					IL_strNCopy(
						SourceStr:= apsElements2[4], 
						DstStr:= ADR(sTemp), 
						CharNum:= 5, 
						strCharFill:= ' ' , 
						MaxLen:= 5);
					{warning 'strNCopy'}					
					//strNCopy(ADR(sTemp), 3, arElements2[4], 3);
		
					//strConcat(ADR(AxesActConfig[k].Firmware), 9, ADR(sTemp));
					IL_CONCAT(ADR(refastAxesActConfig[k].sFirmware), ADR(sTemp), ADR(refastAxesActConfig[k].sFirmware), 9);
					
					//check functional package 
					refastAxesActConfig[k].stFunctionalPackages.bMSP := FALSE;
					refastAxesActConfig[k].stFunctionalPackages.bSRV := FALSE;
					refastAxesActConfig[k].stFunctionalPackages.bSNC := FALSE;
					refastAxesActConfig[k].stFunctionalPackages.bML := FALSE;
					refastAxesActConfig[k].stFunctionalPackages.bMA := FALSE;
					refastAxesActConfig[k].stFunctionalPackages.bTF := FALSE;
					
					IF apsElements2[7]^ = 'MSP' THEN
						refastAxesActConfig[k].stFunctionalPackages.bMSP := TRUE;
					ELSIF apsElements2[7]^ = 'SRV' THEN
						refastAxesActConfig[k].stFunctionalPackages.bSRV := TRUE;
					ELSIF apsElements2[7]^ = 'SNC' THEN
						refastAxesActConfig[k].stFunctionalPackages.bSNC := TRUE;
					END_IF
					
					IF apsElements2[8]^ = 'ML' THEN
						refastAxesActConfig[k].stFunctionalPackages.bML := TRUE;
					ELSIF apsElements2[8]^ = 'MA' THEN
						refastAxesActConfig[k].stFunctionalPackages.bMA := TRUE;
					ELSIF apsElements2[8]^ = 'TF' THEN
						refastAxesActConfig[k].stFunctionalPackages.bTF := TRUE;
					END_IF	
					
					// Check DoubleAxis
					refastAxesActConfig[k].stDoubleAxis.bIsDoubleAxis := FALSE;	
					IF (apsElements2[3]^ = 'MPD') 
						OR (apsElements2[3]^ = 'MPM') THEN		(* 2021-08-03 gt: RDK90 #0124 Placon mit OHNE externe Bremse und neuen Steuerteilen *)
						refastAxesActConfig[k].stDoubleAxis.bIsDoubleAxis := TRUE;
						refastAxesActConfig[k].stDoubleAxis.iLeftAxisAddress := M_GetSercosAdress(apsElements[iMAX_NUM_ELEMENTS_C479*i+4], 1);
						refastAxesActConfig[k].stDoubleAxis.iRightAxisAddress := M_GetSercosAdress(apsElements[iMAX_NUM_ELEMENTS_C479*i+4], 2);
					END_IF
					
					k := k+1;
			
				// no Rexroth IO device and no drive	
				ELSIF NOT (apsElements[iMAX_NUM_ELEMENTS_C479*i+1]^ = '') THEN
					refastSercosIOActConfig[j].bAvailable := TRUE;
					refastSercosIOActConfig[j].iSercosAddress := iSercosAddressTemp;	
	
					//	Präfix noch entfernen !!!
					refastSercosIOActConfig[j].sTypeCode 		:= apsElements[iMAX_NUM_ELEMENTS_C479*i+7]^;
					
					// Where are I/O addresses in C-0-0510
					apiPointerToC510[j] := ADR (aiC510[i+1]);	
					j := j +1;			
				END_IF
			END_IF
		//	i:=i+1;
		//UNTIL( arElements[iMAX_NUM_ELEMENTS_C479*i+1]^ = '' OR i >= MAX_SERCOS_DEVICES )
		//END_REPEAT
		END_FOR

		iState := 50;
		iActNoOfSercosIO := j-1;
		iActNoOfDrives := k-1;
		
		i := 1;
		k := 65;
		j := 0;
		l := 1;


		
(* ################################################################################ *)	
// Sort AxesActConfig by locical address
(* ################################################################################ *)				
	50:
			// real axis configured
			IF aiC484[i] = 8 THEN
				FOR j := 1 TO iMAX_AXES_NUMBER DO
					// if Sercos address is configured copy to temp structure
					IF aiC484[i+1] = refastAxesActConfig[j].iSercosAddress THEN
						astAxesActConfigTmp[(i+1)/2] := refastAxesActConfig[j];
						M_DelStructure(ADR(refastAxesActConfig[j]), SIZEOF(refastAxesActConfig[j]));
						j := iMAX_AXES_NUMBER +1;	// Stop Loop
					END_IF
				END_FOR
			ELSIF  aiC484[i] = 16 THEN
 				astAxesActConfigTmp[(i+1)/2].bVirtualAxis := TRUE;	
			END_IF
						
			IF i < ((2*iMAX_AXES_NUMBER) -1 ) THEN	
				i := i +2;
			ELSE
				FOR j := 1 TO iMAX_AXES_NUMBER DO
					IF refastAxesActConfig[j].bRealAxis THEN
					// Save Sercos Address if drive was found but not configured in C-0-0578	
						refastFoundDrivesError[l].bError := TRUE;
						refastFoundDrivesError[l].iSercosAddress := refastAxesActConfig[j].iSercosAddress;
						refastFoundDrivesError[l].sErrorMessage := 'Axis with sercos adress ';
						sTemp2 := INT_TO_STRING(refastFoundDrivesError[l].iSercosAddress);
						//strConcat(ADR(FoundDrivesError[l].ErrorMessage), SIZEOF(FoundDrivesError[l].ErrorMessage) ,	ADR(strTemp));	
						IL_CONCAT(ADR(refastFoundDrivesError[l].sErrorMessage), ADR(sTemp2), ADR(refastFoundDrivesError[l].sErrorMessage), SIZEOF(refastFoundDrivesError[l].sErrorMessage));				
						sTemp2 := 'found, but not configured with IndraWorks (C-0-0578)';
						//strConcat(ADR	(FoundDrivesError[l].ErrorMessage), SIZEOF(FoundDrivesError[l].ErrorMessage) ,	ADR(strTemp));
						IL_CONCAT(ADR(refastFoundDrivesError[l].sErrorMessage), ADR(sTemp2), ADR(refastFoundDrivesError[l].sErrorMessage), SIZEOF(refastFoundDrivesError[l].sErrorMessage));
						
						IF sDiagMessageInt = '' THEN
							sDiagMessageInt := refastFoundDrivesError[l].sErrorMessage;
						END_IF
						
						ML_SetDiagEntry(
							Severity:= enSeverity, 
							Class:= enClass, 
							Facility:= E_LOG_FACILITY.USER, 
							Code:= wDIAG_CODE, 
							Text:= ADR(refastFoundDrivesError[l].sErrorMessage));
												
						l := l +1;
						bErrorTemp := TRUE;
											
					END_IF
				 	refastAxesActConfig [j] := astAxesActConfigTmp[j];	// copy tmp structure back to origuinal structure
				END_FOR
				iState := 53;
				i := 1;
			END_IF	
		
			IF bErrorTemp THEN
				// If error stop FB
				OUT_ErrorID := 	RESOURCE_ERROR;
				OUT_ErrorIdent.Table :=	USER1_TABLE;       
				OUT_ErrorIdent.Additional1 := 16#F0002;
				OUT_ErrorIdent.Additional2 := 16#F0000;
				
				iState := 998;
			END_IF				

(* ################################################################################ *)	
	// Activate all found axes 
	// necessary to acces S-/P-Parameter
(* ################################################################################ *)	
	53: 
		IF IN_bConfigAxes OR bUpdateFirmware THEN
			REPEAT 	// only new cycle if A24 need to be written
				// activate drive if found on ring
				IF refastAxesActConfig[i].bAvailable THEN 
					stDummyAxis.AxisNo := i;
					iA24 := 0;
					
					IF NOT (iA24 = DWORD_TO_DINT(AxisData[stDummyAxis.AxisNo].dwAxisCondition_i)) THEN		// write A24 only if necessary)
						bExecuteWriteA24 := TRUE;
					END_IF	
				ELSIF aiC484[(2*i)-1] = 8 THEN
					stDummyAxis.AxisNo := i;
					iA24 := 2 ;
					
					IF NOT (iA24 = DWORD_TO_DINT(AxisData[stDummyAxis.AxisNo].dwAxisCondition_i)) THEN		// write A24 only if necessary)
						bExecuteWriteA24 := TRUE;
					END_IF	
				END_IF
						
				fbWriteA24(
					Execute:= bExecuteWriteA24, 
					ParameterNumber:= FP_A_0_0024, 
					Value:= iA24, 
					Axis:= stDummyAxis);	
							
				// NEXT Step
				IF fbWriteA24.Done OR NOT bExecuteWriteA24 THEN	
					bExecuteWriteA24 := FALSE;
					fbWriteA24(
						Execute:= FALSE, 
						Axis:= stDummyAxis );	
					i := i + 1;
				
				// Error	
				ELSIF fbWriteA24.Error THEN
					OUT_ErrorID 	:= fbWriteA24.ErrorID;
					OUT_ErrorIdent 	:= fbWriteA24.ErrorIdent;
					fbWriteA24(Execute	:= FALSE,
								Axis	:= stDummyAxis);
					
					iState 		:= 998;
				END_IF	
			
			
				IF i > iMAX_AXES_NUMBER THEN 
					i := 1;
					iState := 55;
				END_IF
				
			UNTIL bExecuteWriteA24 OR (iState = 55) OR (iState = 998)
			END_REPEAT		
		ELSE
			i := 1;
			iState := 55;
		END_IF
(* ################################################################################ *)	
	// Read name A-0-0002 
(* ################################################################################ *)	
	55:
		REPEAT 	// only new cycle if A-0-0002 needs to be read
			stDummyAxis.AxisNo := i;
		
			bExecuteReadName := (aiC484[2*(i-1)+1] = 8) OR (aiC484[2*(i-1)+1] = 16); // Real (8) and Virtual (16) Axes
			
			fbReadStringParameter(
				Execute:= bExecuteReadName, 
				ParameterNumber:=FP_A_0_0002, 
				Axis:= stDummyAxis, 
				Done=> , 
				Active=> , 
				Error=> , 
				ErrorID=> , 
				ErrorIdent=> , 
				Value=> refastAxesActConfig[i].sName );	
	
			IF NOT fbReadStringParameter.Execute THEN
				refastAxesActConfig[i].sName := '';
			END_IF
				
			IF 	fbReadStringParameter.Done OR NOT bExecuteReadName THEN
				i := i +1 ;
				bExecuteReadName := FALSE;
				
				fbReadStringParameter(
					Execute:= FALSE , 
					ParameterNumber:=FP_A_0_0002 , 
					Axis:= stDummyAxis);
					
				IF i > MB_MAX_AXIS_NUMBER THEN
					i := 1;
					iState := 56;
				END_IF	
				
			ELSIF fbReadStringParameter.Error THEN
					OUT_ErrorID 	:= fbReadStringParameter.ErrorID;
					OUT_ErrorIdent 	:= fbReadStringParameter.ErrorIdent;
					fbReadStringParameter(Execute	:= FALSE,
										Axis	:= stDummyAxis);
					iState 		:= 998;	
			END_IF
	
			
		UNTIL bExecuteReadName OR (iState = 56) OR (iState = 998)
		END_REPEAT	
		
		
(* ################################################################################ *)	
	// Read SerialNo of Drive
(* ################################################################################ *)	
		
	56:
		stDummyAxis.AxisNo := i;
		refastAxesActConfig[i].udiSerialNo := 0;
		
		bExecuteReadSerialNo := (aiC484[2*(i-1)+1] = 8) AND refastAxesActConfig[i].bAvailable;
		
		fbReadListParameter(
			Execute			:= bExecuteReadSerialNo, 
			ParameterNumber	:= GVL_P_Param_ID.FP_P_0_1518, 
			NoOfBytes		:= SIZEOF(audiP1518), 
			ValueAdr		:= ADR(audiP1518), 
			Axis			:= stDummyAxis);	
	
		IF 	fbReadListParameter.Done OR NOT bExecuteReadSerialNo THEN
			IF fbReadListParameter.Done THEN
				refastAxesActConfig[i].udiSerialNo :=	audiP1518[4];	// ELEMENT 4 of P-0-1518
			END_IF
			
			i := i +1 ;
			
			fbReadListParameter(
				Execute:= FALSE , 
				ParameterNumber:= GVL_P_Param_ID.FP_P_0_1518,
				Axis:= stDummyAxis);
				
			IF i >	MB_MAX_AXIS_NUMBER THEN
				i := 1;
				sTemp2 := '';
				iState 		:= 57;
			END_IF	
			
		ELSIF fbReadListParameter.Error THEN
				OUT_ErrorID 	:= fbReadListParameter.ErrorID;
				OUT_ErrorIdent 	:= fbReadListParameter.ErrorIdent;
				fbReadListParameter(Execute	:= FALSE,
									Axis	:= stDummyAxis);
				iState 		:= 998;	
		END_IF

(* ################################################################################ *)	
	// Read Safety Type
(* ################################################################################ *)	
				
	57:
		stDummyAxis.AxisNo := i;
		refastAxesActConfig[i].sSafetyType :=	'';
		sTemp2 := '';
		
		bExecuteReadSafetyType := (aiC484[2*(i-1)+1] = 8) AND refastAxesActConfig[i].bAvailable;
	
		fbReadStringParameter(
			Execute:= bExecuteReadSafetyType , 
			ParameterNumber:= FP_P_0_1520, 
			Axis:= stDummyAxis);	
			
		IF fbReadStringParameter.Done THEN
			sTemp2 := fbReadStringParameter.Value;
		END_IF
						
		IF 	fbReadStringParameter.Done OR NOT bExecuteReadSafetyType THEN
			
			udiNoOfElements := IL_StrSplit(ADR(sTemp2),'-',0,FALSE,ADR(apsElements2),TO_UDINT(SIZEOF(apsElements2) - TO_INT(NOT TO_BOOL(LEN(sTemp2)))) );
		//	IL_StrSplit(ADR(strTemp),'-',0,FALSE,ADR(arElements2),TO_UDINT(SIZEOF(arElements2) - TO_INT(NOT TO_BOOL(LEN(strTemp)))) );
			{warning 'JS: strSplit'}
			//strSplit(ADR(strTemp),CHAR_MINUS,0,FALSE,ADR(arElements));
			 // S4 or L3 or L4 or etc
			IF udiNoOfElements >= 5 THEN 
				refastAxesActConfig[i].sSafetyType  := M_GetSafetyType(apsTypeCodeElements:=apsElements2 , bSecondDoubleAxis:=FALSE );
			ELSE
				refastAxesActConfig[i].sSafetyType  := '';
			END_IF
			
			i := i +1 ;
			sTemp2 := '';
			fbReadStringParameter(
				Execute:= FALSE , 
				ParameterNumber:=FP_P_0_1520 , 
				Axis:= stDummyAxis);
				
			IF i >	MB_MAX_AXIS_NUMBER THEN
				i := 1;	(* 2018-07-03 Kohl: war 0, aber Array mit Index 0 ist nicht zugelassen, deshalb 1 *)
				iState 		:= 59;
			END_IF	
			
		ELSIF fbReadStringParameter.Error THEN
				OUT_ErrorID 	:= fbReadStringParameter.ErrorID;
				OUT_ErrorIdent 	:= fbReadStringParameter.ErrorIdent;
				fbReadStringParameter(Execute	:= FALSE,
									Axis	:= stDummyAxis);
				iState 		:= 998;	
		END_IF
		

(* ################################################################################ *)	
	// Read Firmware directory
(* ################################################################################ *)			
		
//58:
//	// copy to internal variable
//	sFirmwareDirectoryTemp := stDriveFirmwarePath;
//
//	// try to open directory
//	udiDirHandle := SysDirOpen(
//					szDir:=sFirmwareDirectoryTemp , 
//					szDirEntry:= sTemp1, 
//					diMaxDirEntry:= 99  , 
//					pDirInfo:=ADR(ar_stDirInfo) , 
//					pResult:=ADR(udiResultOpen) );
//
//	// directory could be opened 					
//	IF (udiResultOpen = Errors.ERR_OK) THEN
//		// delet structure
//		FOR i := 1 TO MAX_NO_FIRMWARE_FILES DO
//			ar_sFirmwareFiles[i] := '';
//		END_FOR
//		uiNoOfFimrwareFiles := 0;
//		
//		// read all files
//		uiFileNo := 1;
//		udiResultRead := SysDirRead(hDir:=udiDirHandle , szDirEntry:=ar_sFirmwareFiles[uiFileNo] , diMaxDirEntry:= 99, pDirInfo:= 0);
//		REPEAT 
//			udiResultRead := SysDirRead(hDir:=udiDirHandle , szDirEntry:=ar_sFirmwareFiles[uiFileNo] , diMaxDirEntry:= 99, pDirInfo:= 0);
//			
//			//END , no more files available
//			IF (udiResultRead = Errors.ERR_END_OF_OBJECT) THEN
//				ar_sFirmwareFiles[uiFileNo] := '';
//				uiFileNo := uiFileNo -1;
//			ELSE	
//				ar_stFirmwareFilesType[uiFileNo]:=	MO_DUT_funGetFirmwareType(ar_sFirmwareFiles[uiFileNo]);
//				uiFileNo := uiFileNo +1;
//			END_IF	
//			
//		UNTIL (udiResultRead = Errors.ERR_END_OF_OBJECT)
//		END_REPEAT 
//		uiNoOfFirmwareFiles := uiFileNo;
//		SysDirClose(hDir:=udiDirHandle );
//		
//		// finish
//		i := 1;
//		iState 		:= 59;		
//	ELSE	// directory does not exist
//		
//		// create directory
//		udiResutlCreate := SysDirCreate(szDir:=sFirmwareDirectoryTemp);
//		// finish
//		i := 1;
//		iState 		:= 59;		
//	END_IF

(* ################################################################################ *)	
	// Read IP address from drive 
(* ################################################################################ *)			
	59:	
		REPEAT 	// only new cycle if S-0-1020 needs to be read
			stDummyAxis.AxisNo := i;
		
			bExecuteReadName := (aiC484[2*(i-1)+1] = 8) 			// Real (8) 
								AND refastAxesActConfig[i].bAvailable 
								AND (
									(AxisData[stDummyAxis.AxisNo].dwAxisCondition_i = 0)  
									OR (AxisData[stDummyAxis.AxisNo].dwAxisCondition_i = 1) 
									OR (AxisData[stDummyAxis.AxisNo].dwAxisCondition_i = 4) 
									OR (AxisData[stDummyAxis.AxisNo].dwAxisCondition_i = 5)
									OR (AxisData[stDummyAxis.AxisNo].dwAxisCondition_i = 8) 
									OR (AxisData[stDummyAxis.AxisNo].dwAxisCondition_i = 9)
									OR (AxisData[stDummyAxis.AxisNo].dwAxisCondition_i = 12)
									OR (AxisData[stDummyAxis.AxisNo].dwAxisCondition_i = 13)
									);
    
			fbReadListParameter(
				Execute:= bExecuteReadName , 
				ParameterNumber:= FP_S_0_1020 , 
				NoOfBytes:= SIZEOF(abDriveIP) , 
				ValueAdr:= ADR(abDriveIP), 
				Done=> , 
				Active=> , 
				Error=> , 
				ErrorID=> , 
				ErrorIdent=> , 
				NoOfRecBytes=> , 
				Axis:=stDummyAxis );	
							
			IF 	fbReadListParameter.Done OR NOT bExecuteReadName THEN
				IF 	bExecuteReadName THEN			
					refastAxesActConfig[i].sIP := '';
					sTemp2 := BYTE_TO_STRING(abDriveIP[0]) ;
					//strConcat(ADR(AxesActConfig[i].IP), SIZEOF(AxesActConfig[i].IP) ,ADR(strTemp));
					IL_CONCAT(ADR(refastAxesActConfig[i].sIP), ADR(sTemp2), ADR(refastAxesActConfig[i].sIP), SIZEOF(refastAxesActConfig[i].sIP));
					sTemp2 := '.' ;
					IL_CONCAT(ADR(refastAxesActConfig[i].sIP), ADR(sTemp2), ADR(refastAxesActConfig[i].sIP), SIZEOF(refastAxesActConfig[i].sIP));
					sTemp2 := BYTE_TO_STRING(abDriveIP[1]) ;
					IL_CONCAT(ADR(refastAxesActConfig[i].sIP), ADR(sTemp2), ADR(refastAxesActConfig[i].sIP), SIZEOF(refastAxesActConfig[i].sIP));
					sTemp2 := '.' ;
					IL_CONCAT(ADR(refastAxesActConfig[i].sIP), ADR(sTemp2), ADR(refastAxesActConfig[i].sIP), SIZEOF(refastAxesActConfig[i].sIP));
					sTemp2 := BYTE_TO_STRING(abDriveIP[2]) ;
					IL_CONCAT(ADR(refastAxesActConfig[i].sIP), ADR(sTemp2), ADR(refastAxesActConfig[i].sIP), SIZEOF(refastAxesActConfig[i].sIP));
					sTemp2 := '.' ;
					IL_CONCAT(ADR(refastAxesActConfig[i].sIP), ADR(sTemp2), ADR(refastAxesActConfig[i].sIP), SIZEOF(refastAxesActConfig[i].sIP));
					sTemp2 := BYTE_TO_STRING(abDriveIP[3]) ;
					IL_CONCAT(ADR(refastAxesActConfig[i].sIP), ADR(sTemp2), ADR(refastAxesActConfig[i].sIP), SIZEOF(refastAxesActConfig[i].sIP));
				ELSE	
					refastAxesActConfig[i].sIP := '';
				END_IF 
				i := i +1 ;
				bExecuteReadName := FALSE;
				
				fbReadListParameter(
					Execute:= FALSE , 
					ParameterNumber:=FP_S_0_1020 , 
					Axis:= stDummyAxis);
					
				IF i > MB_MAX_AXIS_NUMBER THEN
					i := 0;
					iState := 60;
				END_IF	
				
			ELSIF fbReadListParameter.Error THEN
					OUT_ErrorID 	:= fbReadListParameter.ErrorID;
					OUT_ErrorIdent 	:= fbReadListParameter.ErrorIdent;
					fbReadListParameter(Execute	:= FALSE,
										Axis	:= stDummyAxis);
					iState 		:= 998;	
			END_IF	
		UNTIL bExecuteReadName OR (iState = 60) OR (iState = 998)
		END_REPEAT		
	
		
		
(* ################################################################################ *)	
	// Read ata0b directory
(* ################################################################################ *)			
		
	60:	
		iEntry := 0;
		diMaxEntry := SIZEOF(astDirEntry[iEntry].sEntry);
		Result := SysDirSetCurrent(sPathNameInt);
		hDir := SysDirOpen('', astDirEntry[iEntry].sEntry, diMaxEntry, ADR(dir), ADR(Result));
		iEntry := iEntry + 1;
		WHILE Result = Errors.ERR_OK AND hDir <> RTS_INVALID_HANDLE AND iEntry < iMAX_DIR_ENTRY DO
			diMaxEntry := SIZEOF(astDirEntry[iEntry].sEntry);
			Result := SysDirRead(hDir, astDirEntry[iEntry].sEntry, diMaxEntry, ADR(dir));
			IF (DINT_TO_UDINT(dir.diDirectory) AND DirInfoFlags.DF_DIRECTORY) <> 0 THEN
				astDirEntry[iEntry].bDirectory := TRUE;
			END_IF
			iEntry := iEntry + 1;	
		END_WHILE
		Result := SysDirClose(hDir);
		iEntry := iEntry -2;
		
		
		// create new file or open existing?
		fb_SysFileOpenAsync.stMode := 'rw';

		// 2018-07-03: JK Zählerstart geändert von 1 -> 0, weil im Array schon an der Stelle 0 Informationen stehen		
		FOR i := 0 TO iEntry DO
			IF NOT astDirEntry[i].bDirectory THEN
				IF astDirEntry[i].sEntry = sFILE_NAME THEN
					fb_SysFileOpenAsync.stMode := 'r';
				END_IF
			END_IF
		END_FOR
				
		iState 		:= 65;		
			
		
(* ################################################################################ *)	
	// Open UserDefs.cfg 
(* ################################################################################ *)	
	65:		
		fb_SysFileOpenAsync(
			bEnable:= TRUE, 
			stFileName:= sFILE_AND_PATH, 
			stMode:= , 
			bDone=> , 
			bBusy=> , 
			bError=> , 
			wErrorId=> , 
			hFile=> hCfg);
	
			
		IF fb_SysFileOpenAsync.bDone THEN
			fb_SysFileOpenAsync(
				bEnable:= FALSE);
			sBuffer := '';	
			iState :=70;
		END_IF
	
		// Error	
		IF fb_SysFileOpenAsync.bError THEN
			fb_SysFileOpenAsync(
				bEnable:= FALSE);
			iState :=998;
		END_IF
		
(* ################################################################################ *)	
	// Read UserDefsCfg 
(* ################################################################################ *)	
	70:	// DevicePlcAdd.cfg lesen
		fb_SysFileReadAsync(
			bEnable:= TRUE, 
			hFile:= hCfg, 
			pBuffer:= ADR(sBuffer), 
			dwSize:= INT_TO_DWORD(iFileSize), 
			bDone=> , 
			bBusy=> , 
			bError=> , 
			wErrorId=> , 
			dwRead=> dwReadBytes );
	
		IF fb_SysFileReadAsync.bDone THEN
			fb_SysFileReadAsync(
				bEnable:= FALSE);
			iState := 80;
		END_IF
	
		// Error	
		IF fb_SysFileReadAsync.bError THEN
			fb_SysFileReadAsync(
				bEnable:= FALSE);
			iState :=998;
		END_IF
	
80: // Datei schließen
	fb_SysFileCloseAsync(
		bEnable:= TRUE, 
		hFile:= hCfg, 
		bDone=> , 
		bBusy=> , 
		bError=> , 
		wErrorId=> );

	IF fb_SysFileCloseAsync.bDone THEN
		fb_SysFileCloseAsync(
			bEnable:= FALSE);
		iState :=90;
	END_IF

	// Error	
	IF fb_SysFileCloseAsync.bError THEN
		fb_SysFileCloseAsync(
			bEnable:= FALSE);
		iState :=998;
	END_IF
	
90: // Datei in Array of String kopieren und Formatzeichen löschen
	// split String																//Workaround Defdb00192639, -1 if string is empty					
	udiNoOfElements := IL_StrSplit(ADR(sBuffer),IL_Ascii_to_Char(13),0,FALSE,ADR(apsSplit),TO_UDINT(SIZEOF(apsSplit) - TO_INT(NOT TO_BOOL(LEN(sBuffer)))) ); 
	{warning 'JS: strSplit'}
	//strSplit(ADR(Buffer),13 ,0,FALSE,ADR(arSplit));
	
	sLineFeed := IL_Ascii_to_Char(10);
	iEOF := UDINT_TO_INT(udiNoOfElements);
	
	FOR i := 1 TO UDINT_TO_INT(udiNoOfElements) DO 
		//arStringActCfg[i] := DEL_CHARS(arSplit[i]^, strLineFeed);
		IL_StrTrimAll(SourceStr:=apsSplit[i] , DstStr:=ADR(asStringActCfg[i]) , Char:=sLineFeed , MaxLen:=SIZEOF(apsSplit[i]^)-1 );
	END_FOR
	
	// letzte Zeile löschen
	IF iEOF > 2 THEN
		asStringActCfg[iEOF-1] := ''; 
		iEOF	:= iEOF-2;
	END_IF	
	
	iState := 91;	
	
	
(* ################################################################################ *)	
	// Read Inline IO Config 
(* ################################################################################ *)	
91:	
	fbINLNModuleConfigList(
		Execute:= TRUE, 
		SizeOfModuleConfig:=  SIZEOF(InlineIOCfg), 
		ModuleConfigAdr:= ADR(InlineIOCfg), 
		Done=> , 
		Active=> , 
		Error=> , 
		ErrorID=> , 
		ErrorIdent=> , 
		NoOfModuleConfig=> udiNoOfModuleConfig  );

	
	IF fbINLNModuleConfigList.Done THEN
		FOR i := 1 TO iMAX_INLINE_IO DO	
			IF InlineIOCfg[i].ModuleIdSCN <> 0 THEN
				refastInlineIOActConfig[i].bAvailable := TRUE;
				{warning disable C0196}
				refastInlineIOActConfig[i].eIOType := InlineIOCfg[i].ModuleIdSCN;
				{warning restore C0196}
			END_IF
		END_FOR
		
		fbINLNModuleConfigList(
				Execute:= FALSE );

		i := 1;
		iState := 92;
	ELSIF fbINLNModuleConfigList.Error THEN
		fbINLNModuleConfigList(
				Execute:= FALSE );
		i := 1;		
		iState := 92;
	END_IF

(* ################################################################################ *)	
	// Read S20BK+ ModuleType
(* ################################################################################ *)	
92:	
		stDummyAxis.AxisNo := Objects.SERCOS_ADDRESS_1 + refastSercosIOActConfig[i].iSercosAddress -1;
	
		//SercosIOActConfig[i].TypeCode := DUT_S20Type.S20_UNDEFINED;
		
		// Only with S20 BK+
		bExecuteReadModuleType:= refastSercosIOActConfig[i].bAvailable AND (refastSercosIOActConfig[i].sTypeCode ='R911173318');	
		        
		fbReadListParameter(
			Execute			:= bExecuteReadModuleType, 
			ParameterNumber	:= IL_SIIIElementsToIdn(IL_S_PARAM, 0, 1500, 0, 3),(*= Idn = S-0-1500.0.3*) 			
			NoOfBytes		:= SIZEOF(aliS1500_0_3), 
			ValueAdr		:= ADR(aliS1500_0_3), 
			Axis			:= stDummyAxis);	
	
		IF 	fbReadListParameter.Done OR NOT bExecuteReadModuleType THEN
			IF fbReadListParameter.Done THEN			
				FOR j := 0 TO iMAX_MODULE_ON_SERCOS_IO DO
					refastSercosIOActConfig[i].astIOModule[j].IOType := aliS1500_0_3[j];
					refastSercosIOActConfig[i].astIOModule[j].bAvailable :=  (aliS1500_0_3[j] <> LINT#0);
				END_FOR			
			END_IF
			
			i := i +1 ;	
			fbReadListParameter(
				Execute:= FALSE , 
				Axis:= stDummyAxis);
				
			IF i > iMAX_SERCOS_IO(*MB_MAX_AXIS_NUMBER*) THEN		(* 2018-07-03 Kohl: nun MAX_SERCOS_IO, war MB_MAX_AXIS_NUMBER *)
				i := 1;
				sTemp2 := '';
				iState 		:= 99;
			END_IF	
			
		ELSIF fbReadListParameter.Error THEN
				OUT_ErrorID 	:= fbReadListParameter.ErrorID;
				OUT_ErrorIdent 	:= fbReadListParameter.ErrorIdent;
				fbReadListParameter(Execute	:= FALSE,
									Axis	:= stDummyAxis);
				iState 		:= 998;	
		END_IF

(* ################################################################################ *)	
	// End 
(* ################################################################################ *)	
	99:		
		iState := 100;
			
END_CASE
END_METHOD

METHOD M_1ConfigAxes : BOOL

CASE iState OF

	100:
			IF IN_bCheckAxesConfig AND (IN_bConfigAxes OR bUpdateFirmware) THEN 
				iState := 110;
			ELSIF IN_bConfigAxes OR bUpdateFirmware THEN
				i := 1;
				iState := 120;	
			ELSE
				iState := 199;	
			END_IF

(* ################################################################################ *)	
	// Check drive configuration
(* ################################################################################ *)		
	110:
		FOR i := 1 TO iMAX_AXES_NUMBER DO
			// Reset Error structure
			refastAxesConfigError[i].bWrongSercosAddress			:= FALSE;	
			refastAxesConfigError[i].bWrongFirmware 				:= FALSE;
			refastAxesConfigError[i].bWrongFunctionalPackages 		:= FALSE;
			refastAxesConfigError[i].bWrongDoubleAxisConfiguration := FALSE;
			refastAxesConfigError[i].bWrongSafetyType				:= FALSE;
			refastAxesConfigError[i].bDriveFoundAndNotConfigured 	:= FALSE;
			refastAxesConfigError[i].bDriveConfiguredAndNotFound 	:= FALSE;
		
			// Check if found axis = configured axis
			IF  refastAxesActConfig[i].bRealAxis 
				AND refastAxesActConfig[i].bAvailable 
				AND refastAxesCmdConfig[i].bActive THEN
				IF refastAxesActConfig[i].bRealAxis = refastAxesCmdConfig[i].bRealAxis THEN
					// Sercos Address
					IF NOT (refastAxesActConfig[i].iSercosAddress = refastAxesCmdConfig[i].iSercosAddress) THEN
						refastAxesConfigError[i].bWrongSercosAddress := TRUE;
					END_IF
					// Firmware
					IF NOT (LEFT(refastAxesActConfig[i].sFirmware,6) = refastAxesCmdConfig[i].sFirmware) THEN
						refastAxesConfigError[i].bWrongFirmware := TRUE;	
					END_IF  	
					// Functional Packages	
					IF NOT (refastAxesActConfig[i].stFunctionalPackages.bMA = refastAxesCmdConfig[i].stFunctionalPackages.bMA) 
						OR NOT (refastAxesActConfig[i].stFunctionalPackages.bML = refastAxesCmdConfig[i].stFunctionalPackages.bML)
						OR NOT (refastAxesActConfig[i].stFunctionalPackages.bMSP = refastAxesCmdConfig[i].stFunctionalPackages.bMSP)
						OR NOT (refastAxesActConfig[i].stFunctionalPackages.bSNC = refastAxesCmdConfig[i].stFunctionalPackages.bSNC)
						OR NOT (refastAxesActConfig[i].stFunctionalPackages.bSRV = refastAxesCmdConfig[i].stFunctionalPackages.bSRV)
						OR NOT (refastAxesActConfig[i].stFunctionalPackages.bTF = refastAxesCmdConfig[i].stFunctionalPackages.bTF) 
						OR NOT (refastAxesActConfig[i].stFunctionalPackages.bCL = refastAxesCmdConfig[i].stFunctionalPackages.bCL)
						THEN
							refastAxesConfigError[i].bWrongFunctionalPackages := TRUE;	
					END_IF
					// SafetyType
					IF NOT (refastAxesActConfig[i].sSafetyType = refastAxesCmdConfig[i].sSafetyType) THEN
						refastAxesConfigError[i].bWrongSafetyType := TRUE;	
					END_IF  	
					// Double Axis Configuration
					IF NOT (refastAxesActConfig[i].stDoubleAxis.bIsDoubleAxis = refastAxesCmdConfig[i].stDoubleAxis.bIsDoubleAxis)
					OR (
					( NOT (refastAxesActConfig[i].stDoubleAxis.iLeftAxisAddress = refastAxesCmdConfig[i].stDoubleAxis.iLeftAxisAddress)
					OR  NOT (refastAxesActConfig[i].stDoubleAxis.iRightAxisAddress = refastAxesCmdConfig[i].stDoubleAxis.iRightAxisAddress)	
					) AND refastAxesActConfig[i].stDoubleAxis.bIsDoubleAxis AND refastAxesCmdConfig[i].stDoubleAxis.bIsDoubleAxis 					
						) THEN
						refastAxesConfigError[i].bWrongDoubleAxisConfiguration := TRUE;			
					END_IF
				END_IF
			// Found but not configured	
			ELSIF refastAxesActConfig[i].bRealAxis 
				AND refastAxesActConfig[i].bAvailable 
				AND NOT refastAxesCmdConfig[i].bActive THEN
				refastAxesConfigError[i].bDriveFoundAndNotConfigured := TRUE;
			// configured but not found
			ELSIF refastAxesCmdConfig[i].bRealAxis
				AND NOT refastAxesActConfig[i].bAvailable
				AND refastAxesCmdConfig[i].bActive 
				THEN
				refastAxesConfigError[i].bDriveConfiguredAndNotFound := TRUE;
			END_IF
			
			IF refastAxesConfigError[i].bWrongSercosAddress	
				OR refastAxesConfigError[i].bWrongFirmware 
				OR refastAxesConfigError[i].bWrongSafetyType 
				OR refastAxesConfigError[i].bWrongFunctionalPackages 
				OR refastAxesConfigError[i].bWrongDoubleAxisConfiguration
				OR refastAxesConfigError[i].bDriveFoundAndNotConfigured 
				OR refastAxesConfigError[i].bDriveConfiguredAndNotFound THEN
				refastAxesConfigError[i].bError := TRUE;
				bErrorTemp := TRUE;
				
				// Create Error Message
				refastAxesConfigError[i].sErrorMessage := 'Axis ';
				sTemp2 := refastAxesActConfig[i].sName;
				//strConcat(ADR	(AxesConfigError[i].ErrorMessage), SIZEOF(AxesConfigError[i].ErrorMessage) ,	ADR(strTemp));
				IL_CONCAT(ADR(refastAxesConfigError[i].sErrorMessage), ADR(sTemp2), ADR(refastAxesConfigError[i].sErrorMessage), SIZEOF(refastAxesConfigError[i].sErrorMessage));
				sTemp2 := ' with sercos address ';
				IL_CONCAT(ADR(refastAxesConfigError[i].sErrorMessage), ADR(sTemp2), ADR(refastAxesConfigError[i].sErrorMessage), SIZEOF(refastAxesConfigError[i].sErrorMessage));
				sTemp2 := INT_TO_STRING(refastAxesActConfig[i].iSercosAddress);
				IL_CONCAT(ADR(refastAxesConfigError[i].sErrorMessage), ADR(sTemp2), ADR(refastAxesConfigError[i].sErrorMessage), SIZEOF(refastAxesConfigError[i].sErrorMessage));
				sTemp2 := ' shows following error(s): ';
				IL_CONCAT(ADR(refastAxesConfigError[i].sErrorMessage), ADR(sTemp2), ADR(refastAxesConfigError[i].sErrorMessage), SIZEOF(refastAxesConfigError[i].sErrorMessage));
				sTemp2 :='';
				
				IF refastAxesConfigError[i].bWrongSercosAddress	THEN
					sTemp2 :='wrong sercos address';
					//strConcat(ADR	(AxesConfigError[i].ErrorMessage), SIZEOF(AxesConfigError[i].ErrorMessage) ,	ADR(strTemp));
					IL_CONCAT(ADR(refastAxesConfigError[i].sErrorMessage), ADR(sTemp2), ADR(refastAxesConfigError[i].sErrorMessage), SIZEOF(refastAxesConfigError[i].sErrorMessage));
					sTemp2 :=', ';
				END_IF
					
				IF refastAxesConfigError[i].bWrongFirmware	THEN
					//strConcat(ADR	(AxesConfigError[i].ErrorMessage), SIZEOF(AxesConfigError[i].ErrorMessage) ,	ADR(strTemp));
					IL_CONCAT(ADR(refastAxesConfigError[i].sErrorMessage), ADR(sTemp2), ADR(refastAxesConfigError[i].sErrorMessage), SIZEOF(refastAxesConfigError[i].sErrorMessage));
					sTemp2 :='wrong firmware';
					//strConcat(ADR	(AxesConfigError[i].ErrorMessage), SIZEOF(AxesConfigError[i].ErrorMessage) ,	ADR(strTemp));
					IL_CONCAT(ADR(refastAxesConfigError[i].sErrorMessage), ADR(sTemp2), ADR(refastAxesConfigError[i].sErrorMessage), SIZEOF(refastAxesConfigError[i].sErrorMessage));
					sTemp2 :=', ';
				END_IF
				
				IF refastAxesConfigError[i].bWrongSafetyType	THEN
					//strConcat(ADR	(AxesConfigError[i].ErrorMessage), SIZEOF(AxesConfigError[i].ErrorMessage) ,	ADR(strTemp));
					IL_CONCAT(ADR(refastAxesConfigError[i].sErrorMessage), ADR(sTemp2), ADR(refastAxesConfigError[i].sErrorMessage), SIZEOF(refastAxesConfigError[i].sErrorMessage));
					sTemp2 :='wrong SafetyType';
					//strConcat(ADR	(AxesConfigError[i].ErrorMessage), SIZEOF(AxesConfigError[i].ErrorMessage) ,	ADR(strTemp));
					IL_CONCAT(ADR(refastAxesConfigError[i].sErrorMessage), ADR(sTemp2), ADR(refastAxesConfigError[i].sErrorMessage), SIZEOF(refastAxesConfigError[i].sErrorMessage));
					sTemp2 :=', ';
				END_IF
				
				IF refastAxesConfigError[i].bWrongFunctionalPackages	THEN
					//strConcat(ADR	(AxesConfigError[i].ErrorMessage), SIZEOF(AxesConfigError[i].ErrorMessage) ,	ADR(strTemp));
					IL_CONCAT(ADR(refastAxesConfigError[i].sErrorMessage), ADR(sTemp2), ADR(refastAxesConfigError[i].sErrorMessage), SIZEOF(refastAxesConfigError[i].sErrorMessage));
					sTemp2 :='wrong functional package';
					//strConcat(ADR	(AxesConfigError[i].ErrorMessage), SIZEOF(AxesConfigError[i].ErrorMessage) ,	ADR(strTemp));
					IL_CONCAT(ADR(refastAxesConfigError[i].sErrorMessage), ADR(sTemp2), ADR(refastAxesConfigError[i].sErrorMessage), SIZEOF(refastAxesConfigError[i].sErrorMessage));
					sTemp2 :=', ';
				END_IF
				
				IF refastAxesConfigError[i].bWrongDoubleAxisConfiguration	THEN
					//strConcat(ADR	(AxesConfigError[i].ErrorMessage), SIZEOF(AxesConfigError[i].ErrorMessage) ,	ADR(strTemp));
					IL_CONCAT(ADR(refastAxesConfigError[i].sErrorMessage), ADR(sTemp2), ADR(refastAxesConfigError[i].sErrorMessage), SIZEOF(refastAxesConfigError[i].sErrorMessage));
					sTemp2 :='wrong double axis config';
					//strConcat(ADR	(AxesConfigError[i].ErrorMessage), SIZEOF(AxesConfigError[i].ErrorMessage) ,	ADR(strTemp));
					IL_CONCAT(ADR(refastAxesConfigError[i].sErrorMessage), ADR(sTemp2), ADR(refastAxesConfigError[i].sErrorMessage), SIZEOF(refastAxesConfigError[i].sErrorMessage));
					sTemp2 :=', ';
				END_IF
				
				IF refastAxesConfigError[i].bDriveConfiguredAndNotFound	THEN
					//strConcat(ADR	(AxesConfigError[i].ErrorMessage), SIZEOF(AxesConfigError[i].ErrorMessage) ,	ADR(strTemp));
					IL_CONCAT(ADR(refastAxesConfigError[i].sErrorMessage), ADR(sTemp2), ADR(refastAxesConfigError[i].sErrorMessage), SIZEOF(refastAxesConfigError[i].sErrorMessage));
					sTemp2 :='configured but not found';
					//strConcat(ADR	(AxesConfigError[i].ErrorMessage), SIZEOF(AxesConfigError[i].ErrorMessage) ,	ADR(strTemp));
					IL_CONCAT(ADR(refastAxesConfigError[i].sErrorMessage), ADR(sTemp2), ADR(refastAxesConfigError[i].sErrorMessage), SIZEOF(refastAxesConfigError[i].sErrorMessage));
					sTemp2 :=', ';
				END_IF
				
				IF refastAxesConfigError[i].bDriveFoundAndNotConfigured	THEN
					//strConcat(ADR	(AxesConfigError[i].ErrorMessage), SIZEOF(AxesConfigError[i].ErrorMessage) ,	ADR(strTemp));
					IL_CONCAT(ADR(refastAxesConfigError[i].sErrorMessage), ADR(sTemp2), ADR(refastAxesConfigError[i].sErrorMessage), SIZEOF(refastAxesConfigError[i].sErrorMessage));
					sTemp2 :='found but not configured in DeviceCmdConfig';
					//strConcat(ADR	(AxesConfigError[i].ErrorMessage), SIZEOF(AxesConfigError[i].ErrorMessage) ,	ADR(strTemp));
					IL_CONCAT(ADR(refastAxesConfigError[i].sErrorMessage), ADR(sTemp2), ADR(refastAxesConfigError[i].sErrorMessage), SIZEOF(refastAxesConfigError[i].sErrorMessage));
					sTemp2 :=', ';
				END_IF
					
				ML_SetDiagEntry(
						Severity:= enSeverity, 
						Class:= enClass, 
						Facility:= E_LOG_FACILITY.USER, 
						Code:= wDIAG_CODE, 
						Text:= ADR(refastAxesConfigError[i].sErrorMessage));
						
				IF sDiagMessageInt = '' THEN
					sDiagMessageInt := refastAxesConfigError[i].sErrorMessage;
				END_IF		
			
			END_IF
		END_FOR
		
		IF bErrorTemp THEN
		// If error stop FB
			OUT_ErrorID := 	RESOURCE_ERROR;
			OUT_ErrorIdent.Table :=	USER1_TABLE;       
			OUT_ErrorIdent.Additional1 := 16#F0001;
			OUT_ErrorIdent.Additional2 := 16#F0000;
			
			iState := 998;
		ELSE
		// If no error activate all found drives
			iState := 120;	
			i := 1;
		END_IF
		
(* ################################################################################ *)	
	// Activate all found axes
(* ################################################################################ *)	
	120: 
		REPEAT 		// only new cycle if A24 need to be written
			// activate drive if found on ring
			IF refastAxesActConfig[i].bAvailable THEN 
				stDummyAxis.AxisNo := i;
				CASE refastAxesCmdConfig[i].iStatus OF  			
					0: iA24 := 0;
					1: iA24 := 1;
					2: iA24 := 1;
					
					4: iA24 := 4;
					5: iA24 := 5;
					6: iA24 := 5; 
					
					8: iA24 := 8;
					9: iA24 := 9;
					10: iA24 := 9;
				
					12: iA24 := 12; 
					13: iA24 := 13;
					14: iA24 := 13;
					ELSE
						iA24 := 0;
				END_CASE
				
				IF NOT (iA24 = DWORD_TO_DINT(AxisData[stDummyAxis.AxisNo].dwAxisCondition_i)) THEN		// write A24 only if necessary)
					bExecuteWriteA24 := TRUE;
				END_IF	
			ELSIF aiC484[(2*i)-1] = 8 THEN
				stDummyAxis.AxisNo := i;
				// If drive was not on ring
				IF ((refastAxesCmdConfig[i].iStatus > 3) 
						AND (refastAxesCmdConfig[i].iStatus < 7)) THEN
						//Write A24 if command value decoupling is configured
						iA24 := 6;
				ELSIF ((refastAxesCmdConfig[i].iStatus > 11) 
						AND (refastAxesCmdConfig[i].iStatus < 15)) THEN 
					//Write A24 if command value decoupling is configured in PM
					iA24 := 14;
				ELSIF ((refastAxesCmdConfig[i].iStatus > 7) 
						AND (refastAxesCmdConfig[i].iStatus < 11)) THEN 
					//Deactivate Drive in PM
					iA24 := 10 ;
				ELSIF ((refastAxesCmdConfig[i].iStatus > 0) 
						AND (refastAxesCmdConfig[i].iStatus < 3)) THEN 
					//Deactivate Drive
					iA24 := 2 ;
				ELSE	
					//Deactivate Drive
					iA24 := 2 ;
				END_IF
				
				IF NOT (iA24 = DWORD_TO_DINT(AxisData[stDummyAxis.AxisNo].dwAxisCondition_i)) THEN		// write A24 only if necessary)
					bExecuteWriteA24 := TRUE;
				END_IF	
			END_IF
			
			fbWriteA24(
				Execute:= bExecuteWriteA24, 
				ParameterNumber:= FP_A_0_0024, 
				Value:= iA24, 
				Axis:= stDummyAxis);	
						
			// NEXT Step
			IF fbWriteA24.Done OR NOT bExecuteWriteA24 THEN	
				bExecuteWriteA24 := FALSE;
				fbWriteA24(
					Execute:= FALSE, 
					Axis:= stDummyAxis );	
				i := i + 1;
			
			// Error	
			ELSIF fbWriteA24.Error THEN
				OUT_ErrorID 	:= fbWriteA24.ErrorID;
				OUT_ErrorIdent 	:= fbWriteA24.ErrorIdent;
				fbWriteA24(Execute	:= FALSE,
							Axis	:= stDummyAxis);
				
				iState 		:= 998;
			END_IF	
		
			IF i > iMAX_AXES_NUMBER THEN 
				iState := 130;
			END_IF
			
		UNTIL bExecuteWriteA24 OR (iState = 130) OR (iState = 998)
		END_REPEAT		
130:
(* ################################################################################ *)	
// create String for UserDefs.cfg
(* ################################################################################ *)				
	iLineCfg := 1;
	//	Header
	asStringCmdCfg[iLineCfg] := ';--------------- Sercos IO --------------- ';
	iLineCfg := iLineCfg + 1;	 	// next line
	asStringCmdCfg[iLineCfg] := '[SercosIO.Master.0]';	
	iLineCfg := iLineCfg +1;	 	// next line	
	FOR i := 1 TO iMAX_AXES_NUMBER DO
		IF  refastAxesCmdConfig[i].iSercosAddress <> 0 
		AND (	// Entry only with CSoS Safety Axes
			(refastAxesCmdConfig[i].sSafetyType = 'S0')
		OR 	(refastAxesCmdConfig[i].sSafetyType = 'S4')
		OR 	(refastAxesCmdConfig[i].sSafetyType = 'S5')
		OR 	(refastAxesCmdConfig[i].sSafetyType = 'S6')
		OR 	(refastAxesCmdConfig[i].sSafetyType = 'S3')
		OR 	(refastAxesCmdConfig[i].sSafetyType = 'SD')
			) THEN 
			IF  refastAxesActConfig[i].bAvailable THEN
				asStringCmdCfg[iLineCfg] := '; ';
			ELSE			
				asStringCmdCfg[iLineCfg] := '';
			END_IF	
			
			sTemp2 := 'SlaveDeactAddr = ';
			//strConcat(ADR	(arStringCmdCfg[iLineCfg]), SIZEOF(arStringCmdCfg[iLineCfg]) ,	ADR(strTemp));
			IL_CONCAT(ADR(asStringCmdCfg[iLineCfg]), ADR(sTemp2), ADR(asStringCmdCfg[iLineCfg]), SIZEOF(asStringCmdCfg[iLineCfg]));
			sTemp2 := INT_TO_STRING (refastAxesCmdConfig[i].iSercosAddress);
			//strConcat(ADR	(arStringCmdCfg[iLineCfg]), SIZEOF(arStringCmdCfg[iLineCfg]) ,	ADR(strTemp));
			IL_CONCAT(ADR(asStringCmdCfg[iLineCfg]), ADR(sTemp2), ADR(asStringCmdCfg[iLineCfg]), SIZEOF(asStringCmdCfg[iLineCfg]));

			IF NOT (asStringCmdCfg[iLineCfg]= asStringActCfg[iLineCfg]) THEN
				OUT_bReboot := TRUE;
			END_IF
		
			iLineCfg := iLineCfg +1; 	// next line
		END_IF	
	END_FOR
	// finished
	iState := 199;
	
(* ################################################################################ *)	
	// End
(* ################################################################################ *)			
199: 
	iState := 200;		
	
END_CASE
END_METHOD

METHOD M_2ConfigSercosIO : BOOL

CASE iState OF 

(* ################################################################################ *)	
	// enable SIII Buscoupler 
(* ################################################################################ *)	
	200: 
		M_DelStructure(ADR(sRingString), SIZEOF(sRingString));
		M_DelStructure(ADR(apsElements), SIZEOF(apsElements));	
		M_DelStructure(ADR(refastSercosIOConfigError), SIZEOF(refastSercosIOConfigError));
//		M_DelStructure(ADR(SercosIOCmdConfigError), SIZEOF(SercosIOCmdConfigError));
//		M_DelStructure(ADR(SercosIOActConfig_tmp), SIZEOF(SercosIOActConfig_tmp));	
		M_DelStructure(ADR(abSercosIOFoundInConfig), SIZEOF(abSercosIOFoundInConfig));	
		
		
		IF IN_bConfigSercosIO 
			AND IN_bCheckSercosIOConfig THEN
			iState := 210;			
		ELSIF IN_bConfigSercosIO THEN
			iState := 230;
		ELSIF IN_bCheckSercosIOConfig THEN
			iState := 210;
		ELSIF IN_bWriteSercosIOAddress THEN 
			iState := 290;	
		ELSE
			iState := 299;
		END_IF

(* ################################################################################ *)	
	// validity check if enough IOs are found and configured 
	// Check also correct sercos Adress if WriteSercosIOAddress is not enabled
(* ################################################################################ *)	
	210:
		k := 1;
		bIOFound := FALSE;
		IF NOT IN_bWriteSercosIOAddress THEN
			FOR i := 1 TO iMAX_SERCOS_IO DO	
					
				// Reset Error Struct
				refastSercosIOConfigError[i].bError := FALSE;
				refastSercosIOConfigError[i].sErrorMessage := '';
				refastSercosIOConfigError[i].bIOFoundAndNotConfigured := FALSE;	
				refastSercosIOConfigError[i].bIOConfiguredAndNotFound := FALSE;
				refastSercosIOConfigError[i].bWrongSercosAddress := FALSE;
				refastSercosIOConfigError[i].iSercosAddress := 0;
				refastSercosIOConfigError[i].bWrongIOModuleType := FALSE;
				
				IF NOT (refastSercosIOCmdConfig[i].iSercosAddress = 0) THEN 	
					// search trough ActConfig
					FOR j := 1 TO iMAX_SERCOS_IO DO
						abSercosIOFoundInConfig[i] := FALSE;
						IF refastSercosIOCmdConfig[i].iSercosAddress = refastSercosIOActConfig[j].iSercosAddress THEN
							bIOFound := TRUE;
							abSercosIOFoundInConfig[i] := TRUE;
							astSercosIOActConfigTmp[i] := refastSercosIOActConfig[j];
							IF NOT refastSercosIOCmdConfig[i].bActive AND astSercosIOActConfigTmp[i].bAvailable THEN
		 						refastSercosIOConfigError[i].bIOFoundAndNotConfigured := TRUE;
								refastSercosIOConfigError[i].iSercosAddress := astSercosIOActConfigTmp[i].iSercosAddress;	
								refastSercosIOConfigError[i].sName := '';	
							//ELSIF SercosIOCmdConfig[i].Active AND NOT SercosIOActConfig_tmp[i].Available THEN
							//	SercosIOConfigError[i].IOConfiguredAndNotFound := TRUE;
							ELSIF refastSercosIOCmdConfig[i].bActive AND astSercosIOActConfigTmp[i].bAvailable THEN
								IF IN_bCheckSercosIOModuleConfig THEN
									// Check if number of found modules = configured modules 
									astSercosIOActConfigTmp[i].uiNoOfIO_Modules := 0;	
									refastSercosIOCmdConfig[i].uiNoOfIOModules := 0;	
									FOR k := 1 TO iMAX_MODULE_ON_SERCOS_IO DO
										// Count configured Modules
										IF refastSercosIOCmdConfig[i].astIOModule[k].bActive THEN	
											refastSercosIOCmdConfig[i].uiNoOfIOModules := refastSercosIOCmdConfig[i].uiNoOfIOModules +1;
										END_IF 
										// Count found Modules
										IF astSercosIOActConfigTmp[i].astIOModule[k].bAvailable THEN	
											astSercosIOActConfigTmp[i].uiNoOfIO_Modules := astSercosIOActConfigTmp[i].uiNoOfIO_Modules +1;
										END_IF
									END_FOR
									IF (refastSercosIOCmdConfig[i].uiNoOfIOModules > astSercosIOActConfigTmp[i].uiNoOfIO_Modules) THEN
										refastSercosIOConfigError[i].bMoreIOModulesConfiguredThanFound := TRUE;
										refastSercosIOConfigError[i].iSercosAddress := refastSercosIOCmdConfig[i].iSercosAddress;
										refastSercosIOConfigError[i].sName := refastSercosIOCmdConfig[i].sName;
									ELSIF (astSercosIOActConfigTmp[i].uiNoOfIO_Modules > refastSercosIOCmdConfig[i].uiNoOfIOModules ) THEN
										refastSercosIOConfigError[i].bMoreIOModulesFoundThanConfigured := TRUE;
										refastSercosIOConfigError[i].iSercosAddress := refastSercosIOCmdConfig[i].iSercosAddress;
										refastSercosIOConfigError[i].sName := refastSercosIOCmdConfig[i].sName;
									ELSE
										refastSercosIOConfigError[i].bMoreIOModulesConfiguredThanFound := FALSE;	
										refastSercosIOConfigError[i].bMoreIOModulesFoundThanConfigured := FALSE;		
									END_IF
									
									// IF number of found modules = configured modules check if type is OK
									IF NOT refastSercosIOConfigError[i].bMoreIOModulesConfiguredThanFound AND NOT refastSercosIOConfigError[i].bMoreIOModulesFoundThanConfigured THEN
										l := 0;
										FOR k := 1 TO iMAX_MODULE_ON_SERCOS_IO DO
											IF astSercosIOActConfigTmp[i].astIOModule[k].bAvailable THEN
												l := l+1;
												WHILE (NOT refastSercosIOCmdConfig[i].astIOModule[l].bActive) AND NOT (l = iMAX_MODULE_ON_SERCOS_IO) DO
													l := l+1;
												END_WHILE
												IF NOT (refastSercosIOCmdConfig[i].astIOModule[l].eIOType = astSercosIOActConfigTmp[i].astIOModule[k].IOType) THEN
													refastSercosIOConfigError[i].astIO_Module[l].bWrongIOType := TRUE;
													refastSercosIOConfigError[i].bWrongIOModuleType := TRUE;
													refastSercosIOConfigError[i].iSercosAddress := refastSercosIOCmdConfig[i].iSercosAddress;
													refastSercosIOConfigError[i].sName := refastSercosIOCmdConfig[i].sName;
												ELSE	
													refastSercosIOConfigError[i].astIO_Module[l].bWrongIOType := FALSE;	
												END_IF
											END_IF
										END_FOR
									END_IF
								END_IF	
							END_IF
							j := iMAX_SERCOS_IO + 1; // Loop END
						END_IF
					END_FOR
					
					// if not found in ActConfig
					IF NOT bIOFound AND refastSercosIOCmdConfig[i].bActive THEN
						refastSercosIOConfigError[i].bIOConfiguredAndNotFound := TRUE;
						refastSercosIOConfigError[i].iSercosAddress := refastSercosIOCmdConfig[i].iSercosAddress;
						refastSercosIOConfigError[i].sName := refastSercosIOCmdConfig[i].sName;	
					END_IF
					bIOFound := FALSE;
				END_IF	
			END_FOR
		END_IF

		// to have same index like SercosIOCmdConfig
		FOR i := 1 TO iMAX_SERCOS_IO DO
			refastSercosIOActConfig[i] := astSercosIOActConfigTmp[i];
		END_FOR
		
		iState := 220;	

(* ################################################################################ *)	
	// generate Error if necessary 
(* ################################################################################ *)	
	220:
		FOR i := 1 TO iMAX_SERCOS_IO DO
			IF refastSercosIOConfigError[i].bWrongSercosAddress	
				OR refastSercosIOConfigError[i].bIOFoundAndNotConfigured 
				OR refastSercosIOConfigError[i].bIOConfiguredAndNotFound 
				OR refastSercosIOConfigError[i].bMoreIOModulesConfiguredThanFound
				OR refastSercosIOConfigError[i].bMoreIOModulesFoundThanConfigured	 
				OR refastSercosIOConfigError[i].bWrongIOModuleType THEN
					refastSercosIOConfigError[i].bError := TRUE;
									
					bErrorTemp := TRUE;
									
					// Create Error Message
					refastSercosIOConfigError[i].sErrorMessage := 'sercos IO ';
					sTemp2 := refastSercosIOConfigError[i].sName ;
					//strConcat(ADR	(SercosIOConfigError[i].ErrorMessage), SIZEOF(SercosIOConfigError[i].ErrorMessage) ,	ADR(strTemp));
					IL_CONCAT(ADR(refastSercosIOConfigError[i].sErrorMessage), ADR(sTemp2), ADR(refastSercosIOConfigError[i].sErrorMessage), SIZEOF(refastSercosIOConfigError[i].sErrorMessage));
					sTemp2 :=  ' with address '; ;
					//strConcat(ADR	(SercosIOConfigError[i].ErrorMessage), SIZEOF(SercosIOConfigError[i].ErrorMessage) ,	ADR(strTemp));
					IL_CONCAT(ADR(refastSercosIOConfigError[i].sErrorMessage), ADR(sTemp2), ADR(refastSercosIOConfigError[i].sErrorMessage), SIZEOF(refastSercosIOConfigError[i].sErrorMessage));
					sTemp2 := INT_TO_STRING(refastSercosIOConfigError[i].iSercosAddress);
					//strConcat(ADR	(SercosIOConfigError[i].ErrorMessage), SIZEOF(SercosIOConfigError[i].ErrorMessage) ,	ADR(strTemp));
					IL_CONCAT(ADR(refastSercosIOConfigError[i].sErrorMessage), ADR(sTemp2), ADR(refastSercosIOConfigError[i].sErrorMessage), SIZEOF(refastSercosIOConfigError[i].sErrorMessage));
					sTemp2 := ' shows error: ';
					//strConcat(ADR	(SercosIOConfigError[i].ErrorMessage), SIZEOF(SercosIOConfigError[i].ErrorMessage) ,	ADR(strTemp));
					IL_CONCAT(ADR(refastSercosIOConfigError[i].sErrorMessage), ADR(sTemp2), ADR(refastSercosIOConfigError[i].sErrorMessage), SIZEOF(refastSercosIOConfigError[i].sErrorMessage));
					sTemp2 :='';
					IF refastSercosIOConfigError[i].bWrongSercosAddress	THEN
						sTemp2 :='wrong sercos address';
						//strConcat(ADR	(SercosIOConfigError[i].ErrorMessage), SIZEOF(SercosIOConfigError[i].ErrorMessage) ,	ADR(strTemp));
						IL_CONCAT(ADR(refastSercosIOConfigError[i].sErrorMessage), ADR(sTemp2), ADR(refastSercosIOConfigError[i].sErrorMessage), SIZEOF(refastSercosIOConfigError[i].sErrorMessage));
						sTemp2 :=', ';
					END_IF
					
					IF refastSercosIOConfigError[i].bIOConfiguredAndNotFound	THEN
						//strConcat(ADR	(SercosIOConfigError[i].ErrorMessage), SIZEOF(SercosIOConfigError[i].ErrorMessage) ,	ADR(strTemp));
						IL_CONCAT(ADR(refastSercosIOConfigError[i].sErrorMessage), ADR(sTemp2), ADR(refastSercosIOConfigError[i].sErrorMessage), SIZEOF(refastSercosIOConfigError[i].sErrorMessage));
						sTemp2 :='configured but not found';
						//strConcat(ADR	(SercosIOConfigError[i].ErrorMessage), SIZEOF(SercosIOConfigError[i].ErrorMessage) ,	ADR(strTemp));
						IL_CONCAT(ADR(refastSercosIOConfigError[i].sErrorMessage), ADR(sTemp2), ADR(refastSercosIOConfigError[i].sErrorMessage), SIZEOF(refastSercosIOConfigError[i].sErrorMessage));
						sTemp2 :=', ';
					END_IF
					
					IF refastSercosIOConfigError[i].bIOFoundAndNotConfigured	THEN
						//strConcat(ADR	(SercosIOConfigError[i].ErrorMessage), SIZEOF(SercosIOConfigError[i].ErrorMessage) ,	ADR(strTemp));
						IL_CONCAT(ADR(refastSercosIOConfigError[i].sErrorMessage), ADR(sTemp2), ADR(refastSercosIOConfigError[i].sErrorMessage), SIZEOF(refastSercosIOConfigError[i].sErrorMessage));
						sTemp2 :='found but not configured in DeviceCmdConfig';
						//strConcat(ADR	(SercosIOConfigError[i].ErrorMessage), SIZEOF(SercosIOConfigError[i].ErrorMessage) ,	ADR(strTemp));
						IL_CONCAT(ADR(refastSercosIOConfigError[i].sErrorMessage), ADR(sTemp2), ADR(refastSercosIOConfigError[i].sErrorMessage), SIZEOF(refastSercosIOConfigError[i].sErrorMessage));
						sTemp2 :=', ';
					END_IF	
									
					IF refastSercosIOConfigError[i].bMoreIOModulesConfiguredThanFound THEN
						//strConcat(ADR	(SercosIOConfigError[i].ErrorMessage), SIZEOF(SercosIOConfigError[i].ErrorMessage) ,	ADR(strTemp));
						IL_CONCAT(ADR(refastSercosIOConfigError[i].sErrorMessage), ADR(sTemp2), ADR(refastSercosIOConfigError[i].sErrorMessage), SIZEOF(refastSercosIOConfigError[i].sErrorMessage));
						sTemp2 :='more IO Modules configured than found';
						//strConcat(ADR	(SercosIOConfigError[i].ErrorMessage), SIZEOF(SercosIOConfigError[i].ErrorMessage) ,	ADR(strTemp));
						IL_CONCAT(ADR(refastSercosIOConfigError[i].sErrorMessage), ADR(sTemp2), ADR(refastSercosIOConfigError[i].sErrorMessage), SIZEOF(refastSercosIOConfigError[i].sErrorMessage));
						sTemp2 :=', ';
					END_IF	
					
					IF refastSercosIOConfigError[i].bMoreIOModulesFoundThanConfigured THEN
						//strConcat(ADR	(SercosIOConfigError[i].ErrorMessage), SIZEOF(SercosIOConfigError[i].ErrorMessage) ,	ADR(strTemp));
						IL_CONCAT(ADR(refastSercosIOConfigError[i].sErrorMessage), ADR(sTemp2), ADR(refastSercosIOConfigError[i].sErrorMessage), SIZEOF(refastSercosIOConfigError[i].sErrorMessage));
						sTemp2 :='less IO Modules configured than found';
						//strConcat(ADR	(SercosIOConfigError[i].ErrorMessage), SIZEOF(SercosIOConfigError[i].ErrorMessage) ,	ADR(strTemp));
						IL_CONCAT(ADR(refastSercosIOConfigError[i].sErrorMessage), ADR(sTemp2), ADR(refastSercosIOConfigError[i].sErrorMessage), SIZEOF(refastSercosIOConfigError[i].sErrorMessage));
						sTemp2 :=', ';
					END_IF	
					
					IF refastSercosIOConfigError[i].bWrongIOModuleType THEN
						//'wrong IO Module Type: Module 1: expected SSDIxxx - found: SSDOxx ';
						FOR j := 1 TO iMAX_MODULE_ON_SERCOS_IO DO
							IF refastSercosIOConfigError[i].astIO_Module[j].bWrongIOType THEN
								//strConcat(ADR	(SercosIOConfigError[i].ErrorMessage), SIZEOF(SercosIOConfigError[i].ErrorMessage) ,	ADR(strTemp));
								IL_CONCAT(ADR(refastSercosIOConfigError[i].sErrorMessage), ADR(sTemp2), ADR(refastSercosIOConfigError[i].sErrorMessage), SIZEOF(refastSercosIOConfigError[i].sErrorMessage));
								sTemp2 :='wrong IO Module Type: Module ';
								//strConcat(ADR	(SercosIOConfigError[i].ErrorMessage), SIZEOF(SercosIOConfigError[i].ErrorMessage) ,	ADR(strTemp));
								IL_CONCAT(ADR(refastSercosIOConfigError[i].sErrorMessage), ADR(sTemp2), ADR(refastSercosIOConfigError[i].sErrorMessage), SIZEOF(refastSercosIOConfigError[i].sErrorMessage));
								sTemp2 := INT_TO_STRING (j);
								//strConcat(ADR	(SercosIOConfigError[i].ErrorMessage), SIZEOF(SercosIOConfigError[i].ErrorMessage) ,	ADR(strTemp));
								IL_CONCAT(ADR(refastSercosIOConfigError[i].sErrorMessage), ADR(sTemp2), ADR(refastSercosIOConfigError[i].sErrorMessage), SIZEOF(refastSercosIOConfigError[i].sErrorMessage));
								sTemp2 :=': expected: ';
								//strConcat(ADR	(SercosIOConfigError[i].ErrorMessage), SIZEOF(SercosIOConfigError[i].ErrorMessage) ,	ADR(strTemp));
								IL_CONCAT(ADR(refastSercosIOConfigError[i].sErrorMessage), ADR(sTemp2), ADR(refastSercosIOConfigError[i].sErrorMessage), SIZEOF(refastSercosIOConfigError[i].sErrorMessage));
								sTemp2 := M_S20TypeToString(refastSercosIOCmdConfig[i].astIOModule[j].eIOType);
								//strConcat(ADR	(SercosIOConfigError[i].ErrorMessage), SIZEOF(SercosIOConfigError[i].ErrorMessage) ,	ADR(strTemp));
								IL_CONCAT(ADR(refastSercosIOConfigError[i].sErrorMessage), ADR(sTemp2), ADR(refastSercosIOConfigError[i].sErrorMessage), SIZEOF(refastSercosIOConfigError[i].sErrorMessage));
								sTemp2 :=' - found: ';
								//strConcat(ADR	(SercosIOConfigError[i].ErrorMessage), SIZEOF(SercosIOConfigError[i].ErrorMessage) ,	ADR(strTemp));
								IL_CONCAT(ADR(refastSercosIOConfigError[i].sErrorMessage), ADR(sTemp2), ADR(refastSercosIOConfigError[i].sErrorMessage), SIZEOF(refastSercosIOConfigError[i].sErrorMessage));
								sTemp2 := M_S20TypeToString(refastSercosIOActConfig[i].astIOModule[j].IOType);
								//strConcat(ADR	(SercosIOConfigError[i].ErrorMessage), SIZEOF(SercosIOConfigError[i].ErrorMessage) ,	ADR(strTemp));
								IL_CONCAT(ADR(refastSercosIOConfigError[i].sErrorMessage), ADR(sTemp2), ADR(refastSercosIOConfigError[i].sErrorMessage), SIZEOF(refastSercosIOConfigError[i].sErrorMessage));
								sTemp2 :=', ';
							END_IF
						END_FOR
					END_IF	
					
					ML_SetDiagEntry(
						Severity:= enSeverity, 
						Class:= enClass, 
						Facility:= E_LOG_FACILITY.USER, 
						Code:= wDIAG_CODE, 
						Text:= ADR(refastSercosIOConfigError[i].sErrorMessage));
					
					IF sDiagMessageInt = '' THEN
						sDiagMessageInt := refastSercosIOConfigError[i].sErrorMessage;
					END_IF			
						
			END_IF
		END_FOR
			
		IF bErrorTemp THEN  
			OUT_ErrorID := 	RESOURCE_ERROR;
			OUT_ErrorIdent.Table :=	USER1_TABLE;       
			OUT_ErrorIdent.Additional1 := 16#F0003;
			OUT_ErrorIdent.Additional2 := 16#F0000;

			iState 		:= 998;
		ELSIF IN_bConfigSercosIO THEN
			iState 		:= 230;
		ELSIF IN_bWriteSercosIOAddress THEN 
			iState 		:= 290;
		ELSE	
			iState 		:= 299;
		END_IF		
		
		
		
(* ################################################################################ *)	
	// validity check if IO config in C-0-0478 matches to SercosIOCmdConfig
(* ################################################################################ *)		
	230:
		j:= 1;
	
		FOR i := 1 TO iMAX_SERCOS_IO DO
			IF refastSercosIOActConfigC578[i].bAvailable AND (refastSercosIOCmdConfig[i].iSercosAddress <> 0) THEN
				; // OK
				bLoopEnd := FALSE;
				REPEAT
					IF j <= iMAX_SERCOS_IO THEN
						IF refastSercosIOActConfig[i].bAvailable AND refastSercosIOCmdConfig[j].bActive THEN
							astSercosIOActConfigTmp[j].sName := refastSercosIOCmdConfig[j].sName;
							astSercosIOActConfigTmp[j].sTypeCode := refastSercosIOActConfig[i].sTypeCode;
							astSercosIOActConfigTmp[j].astIOModule := refastSercosIOActConfig[i].astIOModule;
							astSercosIOActConfigTmp[j].bAvailable := TRUE;
							astSercosIOActConfigTmp[j].iSercosAddress := refastSercosIOCmdConfig[j].iSercosAddress;
							j := j+1;
							bLoopend := TRUE;
						ELSIF refastSercosIOActConfig[i].bAvailable AND NOT refastSercosIOCmdConfig[j].bActive THEN
							astSercosIOActConfigTmp[j].sName := refastSercosIOCmdConfig[j].sName;
							//SercosIOActConfig_tmp[j].TypeCode := SercosIOActConfig[j].TypeCode;
							astSercosIOActConfigTmp[j].sTypeCode := '';
							astSercosIOActConfigTmp[j].bAvailable := FALSE;
							astSercosIOActConfigTmp[j].iSercosAddress := refastSercosIOCmdConfig[j].iSercosAddress;
							j := j+1;
						ELSIF NOT refastSercosIOActConfig[i].bAvailable AND (refastSercosIOCmdConfig[j].iSercosAddress <> 0) THEN 
							astSercosIOActConfigTmp[j].sName := refastSercosIOCmdConfig[j].sName;
							//SercosIOActConfig_tmp[j].TypeCode := SercosIOActConfig[j].TypeCode;
							astSercosIOActConfigTmp[j].sTypeCode := '';
							astSercosIOActConfigTmp[j].bAvailable := FALSE;
							astSercosIOActConfigTmp[j].iSercosAddress := refastSercosIOCmdConfig[j].iSercosAddress;
							j := j+1;
						ELSE	
							j := j+1;
						END_IF
					ELSE	
						bLoopEnd := TRUE;
					END_IF	
				UNTIL bLoopEnd
				END_REPEAT
				
//			ELSIF NOT	SercosIOActConfigC578[i].Available AND (SercosIOCmdConfig[i].SercosAddress <> 0) THEN
//				; // Too many IO configured in DeviceCmdConfig.sercos_IO
//				SercosIOCmdConfigError.Error := TRUE;
//				SercosIOCmdConfigError.TooManyIOConfigured := TRUE; 
//				SercosIOCmdConfigError.SercosAddress := SercosIOCmdConfig[i].SercosAddress;
//				SercosIOCmdConfigError.Name := SercosIOCmdConfig[i].Name;
//				SercosIOCmdConfigError.ErrorMessage := 'Too many IO stations configured in DeviceCmdConfig.sercos_IO';
//				i := MAX_SERCOS_IO +1; // end loop
//			ELSIF SercosIOActConfigC578[i].Available AND (SercosIOCmdConfig[i].SercosAddress = 0) THEN	
//				; // Too less IO configured in DeviceCmdConfig.sercos_IO
//				SercosIOCmdConfigError.Error := TRUE;
//				SercosIOCmdConfigError.TooLessIOConfigured := TRUE; 
//				SercosIOCmdConfigError.SercosAddress := SercosIOActConfigC578[i].SercosAddress;
//				SercosIOCmdConfigError.ErrorMessage := 'Too less IO stations configured in DeviceCmdConfig.sercos_IO';
//				i := MAX_SERCOS_IO +1; // end loop
			END_IF
			
			// Write Message to MLC Log
//			IF SercosIOCmdConfigError.Error THEN
//				bError_temp := TRUE;	
//				ML_SetDiagEntry(
//					Severity:= enSeverity, 
//					Class:= enClass, 
//					Facility:= E_LOG_FACILITY.USER, 
//					Code:= wDiagCode, 
//					Text:= ADR(SercosIOCmdConfigError.ErrorMessage));
//					
//				IF strDiagMessage_int = '' THEN
//					strDiagMessage_int := SercosIOCmdConfigError.ErrorMessage;
//				END_IF			
//	
//			END_IF
		END_FOR
	
		IF bErrorTemp THEN  
			OUT_ErrorID := 	RESOURCE_ERROR;
			OUT_ErrorIdent.Table :=	USER1_TABLE;       
			OUT_ErrorIdent.Additional1 := 16#F0004;
			OUT_ErrorIdent.Additional2 := 16#F0000;
			iState 		:= 998;
		ELSE	
			M_DelStructure(ADR(refastSercosIOActConfig), SIZEOF(refastSercosIOActConfig));	
			FOR i := 1 TO iMAX_SERCOS_IO DO
				refastSercosIOActConfig[i] := astSercosIOActConfigTmp[i];
			END_FOR
	
			iState 		:= 280;
		END_IF		


(* ################################################################################ *)	
	// Read actual configuration C-0-0578
(* ################################################################################ *)

		
(*		
(* ################################################################################ *)	
	// Read actual configuration C-0-0578
(* ################################################################################ *)			
	235:
		fbReadListParameter(
			Execute			:= TRUE, 
			ParameterNumber	:= GVL_C_Param_ID.FP_C_0_0578, 
			NoOfBytes		:= SIZEOF(sRingString), 
			ValueAdr		:= ADR(sRingString), 
			Axis			:= NoAxis);
			
			IF fbReadListParameter.Done THEN
				fbReadListParameter(Execute	:= FALSE,
									Axis	:= NoAxis);
				iState 	:= 240;
				strSplit(ADR(sRingString),CHAR_COMMA,0,FALSE,ADR(apsElements));
				i 		:= -1;
			ELSIF fbReadListParameter.Error THEN
				ErrorID 	:= fbReadListParameter.ErrorID;
				ErrorIdent 	:= fbReadListParameter.ErrorIdent;
				fbReadListParameter(Execute	:= FALSE,
									Axis	:= NoAxis);
				iState 		:= 998;
			END_IF
		
(* ################################################################################ *)	
	// insert Buscoupler to C-0-0578
(* ################################################################################ *)		
	240:
		REPEAT
			i:= i+1;
				{warning 'weitere R911 Nummern müssen agelegt werden'}
		UNTIL (FUN_TypeCodeIsRexrothIO(TypeCode:=LEFT (apsElements.arWords[uiNumOfElementC578*i+3]^,13)) OR (apsElements.arWords[uiNumOfElementC578*i+3]^ = ''))  
		END_REPEAT
				
		IF i > 0 THEN
			FOR j := 1 TO i DO
				// Build STRING for 1 Axis 
				arAxisString[j] := '';
				// Comma 
				strComma := ',';
				
				//combine Elemenst to C-0-0578
				// example A94,L03100,L05R911173318,'-',NPLC1_E4,S0x00000000,O0x00000008,V94
				//Ax
				strConcat(ADR(arAxisString[j]), SIZEOF(arAxisString[j]), apsElements.arWords[uiNumOfElementC578*(j-1)+1]);
				strConcat(ADR(arAxisString[j]), SIZEOF(arAxisString[j]), ADR(strComma));
				// L03x
				strConcat(ADR(arAxisString[j]), SIZEOF(arAxisString[j]), apsElements.arWords[uiNumOfElementC578*(j-1)+2]);
				strConcat(ADR(arAxisString[j]), SIZEOF(arAxisString[j]), ADR(strComma));
				// L05x
				strConcat(ADR(arAxisString[j]), SIZEOF(arAxisString[j]), apsElements.arWords[uiNumOfElementC578*(j-1)+3]);
				strConcat(ADR(arAxisString[j]), SIZEOF(arAxisString[j]), ADR(strComma));
				// -
				strConcat(ADR(arAxisString[j]), SIZEOF(arAxisString[j]), apsElements.arWords[uiNumOfElementC578*(j-1)+4]);
				strConcat(ADR(arAxisString[j]), SIZEOF(arAxisString[j]), ADR(strComma));
				// Nx
				strConcat(ADR(arAxisString[j]), SIZEOF(arAxisString[j]), apsElements.arWords[uiNumOfElementC578*(j-1)+5]);
				strConcat(ADR(arAxisString[j]), SIZEOF(arAxisString[j]), ADR(strComma));
				// S0x
				strConcat(ADR(arAxisString[j]), SIZEOF(arAxisString[j]), apsElements.arWords[uiNumOfElementC578*(j-1)+6]);
				strConcat(ADR(arAxisString[j]), SIZEOF(arAxisString[j]), ADR(strComma));
				// O0x
				strConcat(ADR(arAxisString[j]), SIZEOF(arAxisString[j]), apsElements.arWords[uiNumOfElementC578*(j-1)+7]);
				strConcat(ADR(arAxisString[j]), SIZEOF(arAxisString[j]), ADR(strComma));
				// Vx
				strConcat(ADR(arAxisString[j]), SIZEOF(arAxisString[j]), apsElements.arWords[uiNumOfElementC578*(j-1)+8]);
			
			END_FOR
		END_IF	
		
		k := i+1;
		i := i -1;

		iState := 250;
		
(* ################################################################################ *)	
	// Build Axis/Buscoupler strings 
(* ################################################################################ *)			
	250:
		// how many buscoupler in C578?	
		REPEAT
			i:= i+1;
		UNTIL (apsElements.arWords[uiNumOfElementC578*i+3]^ = '')  
		END_REPEAT
	
				
		FOR j := k TO i DO   
				//Delete 'A' at beginning of String
			IF (apsElements.arWords[uiNumOfElementC578*(j-1)+1]^ <> '') THEN
				ptString := apsElements.arWords[uiNumOfElementC578*(j-1)+1]+1;
			ELSE
				ptString := apsElements.arWords[uiNumOfElementC578*(j-1)+1];
			END_IF
			
			iSercosAddressTemp :=  STRING_TO_INT(ptString^);	
			
			// Check if IO in SercosIOCmdConfig and set Status depending SercosIOCmdConfig.Active
			FOR l := 1 TO MAX_SERCOS_IO DO
				IF SercosIOCmdConfig[l].SercosAddress = iSercosAddressTemp THEN
					// Build String for C578	
					arAxisString[j] := '';
					// Comma 
					strComma := ',';
	
					//combine Elemenst to C-0-0578
					// example A94,L03100,L05R911173318,'-',NPLC1_E4,S0x00000000,O0x00000008,V94
					//Ax
					strConcat(ADR(arAxisString[j]), SIZEOF(arAxisString[j]), apsElements.arWords[uiNumOfElementC578*(j-1)+1]);
					strConcat(ADR(arAxisString[j]), SIZEOF(arAxisString[j]), ADR(strComma));
					// L03x
					strConcat(ADR(arAxisString[j]), SIZEOF(arAxisString[j]), apsElements.arWords[uiNumOfElementC578*(j-1)+2]);
					strConcat(ADR(arAxisString[j]), SIZEOF(arAxisString[j]), ADR(strComma));
					// L05x
					strConcat(ADR(arAxisString[j]), SIZEOF(arAxisString[j]), apsElements.arWords[uiNumOfElementC578*(j-1)+3]);
					strConcat(ADR(arAxisString[j]), SIZEOF(arAxisString[j]), ADR(strComma));
					// -
					strConcat(ADR(arAxisString[j]), SIZEOF(arAxisString[j]), apsElements.arWords[uiNumOfElementC578*(j-1)+4]);
					strConcat(ADR(arAxisString[j]), SIZEOF(arAxisString[j]), ADR(strComma));
					// N
					strConcat(ADR(arAxisString[j]), SIZEOF(arAxisString[j]), apsElements.arWords[uiNumOfElementC578*(j-1)+5]);
					strConcat(ADR(arAxisString[j]), SIZEOF(arAxisString[j]), ADR(strComma));
					// Status
					IF SercosIOCmdConfig[l].Active THEN
						strTemp := 'S0x00000000';
					ELSE
						strTemp := 'S0x00000002';
					END_IF
					strConcat(ADR(arAxisString[j]), SIZEOF(arAxisString[j]), ADR(strTemp));
					strConcat(ADR(arAxisString[j]), SIZEOF(arAxisString[j]), ADR(strComma));
					// 0Ox
					strConcat(ADR(arAxisString[j]), SIZEOF(arAxisString[j]), apsElements.arWords[uiNumOfElementC578*(j-1)+7]);
					strConcat(ADR(arAxisString[j]), SIZEOF(arAxisString[j]), ADR(strComma));
					// Vx
					strConcat(ADR(arAxisString[j]), SIZEOF(arAxisString[j]), apsElements.arWords[uiNumOfElementC578*(j-1)+5]);
				END_IF
				// End LOOP
				IF SercosIOCmdConfig[l].SercosAddress = 0 THEN 
					l := MAX_SERCOS_IO + 1;
				END_IF
			END_FOR
			
		END_FOR
	
		j := j-1;
		iState := 260;

(* ################################################################################ *)	
	// Build C-0-0578 
(* ################################################################################ *)			
	260:	
		//BUILD C-0-0478
		strC578 :='';
		
		IF j > 0 THEN 
			FOR i := 1 TO j DO
				IF i < j THEN
					strConcat(ADR(strC578), (SIZEOF(strC578)), ADR(arAxisString[i]));
					strConcat(ADR(strC578), (SIZEOF(strC578)), ADR(strComma));
				ELSE	
					strConcat(ADR(strC578), (SIZEOF(strC578)), ADR(arAxisString[i]));
				END_IF
			END_FOR
		END_IF

		iState := 270;


(* ################################################################################ *)	
	// Write C-0-0478
(* ################################################################################ *)			
	270: 
		iState := 280;	
	//	WriteC578(
	//		Execute:= TRUE, 
	//		ParameterNumber:= FP_C_0_0578, 
	//		NoOfBytes:= SIZEOF(strC578), 
	//		ValueAdr:= ADR(strC578), 
	//		Axis:= NoAxis, 
	//		Done=> , 
	//		Active=> );
    //
	//	IF WriteC578.Done THEN
	//		WriteC578(Execute	:= FALSE,
	//				Axis	:= NoAxis);
	//		i		:= 0;
	//				
	//
	//	ELSIF WriteC578.Error THEN
	//		ErrorID 	:= WriteC578.ErrorID;
	//		ErrorIdent 	:= WriteC578.ErrorIdent;
	//		WriteC578(Execute	:= FALSE,
	//							Axis	:= NoAxis);
	//		iState 		:= 998;
	//	END_IF
						
*)		
(* ################################################################################ *)	
// create String for UserDefs.cfg
(* ################################################################################ *)						
	280:
		(* Example:
		;---------- Master.0 ----------
		[SercosIO.Master.0]
		SlaveDeactAddr = 20
		SlaveDeactAddr = 32
		SlaveDeactAddr = 35
		SlaveDeactAddr = 56
		SlaveAddr = 40, DeactModule= 2, 4
		SlaveAddr = 55, DeactLastModules= 3

		;------------------------------
		*)
		IF NOT (iLineCfg > 1) THEN
			//	Header
			asStringCmdCfg[iLineCfg] := ';--------------- Sercos IO --------------- ';
			iLineCfg := iLineCfg + 1;	 	// next line
			asStringCmdCfg[iLineCfg] := '[SercosIO.Master.0]';	
			iLineCfg := iLineCfg +1;	 	// next line
		END_IF
		FOR i := 1 TO iMAX_SERCOS_IO DO
			IF refastSercosIOCmdConfig[i].iSercosAddress <> 0 THEN 
				// deactivate only modules
				IF refastSercosIOCmdConfig[i].bActive THEN
					asStringCmdCfg[iLineCfg] := '';
					bWriteThisLine := FALSE;
					sTemp2 := 'SlaveAddr = ';
					//strConcat(ADR	(arStringCmdCfg[iLineCfg]), SIZEOF(arStringCmdCfg[iLineCfg]) ,	ADR(strTemp));
					IL_CONCAT(ADR(asStringCmdCfg[iLineCfg]), ADR(sTemp2), ADR(asStringCmdCfg[iLineCfg]), SIZEOF(asStringCmdCfg[iLineCfg]));
					sTemp2 := INT_TO_STRING (refastSercosIOCmdConfig[i].iSercosAddress);
					//strConcat(ADR	(arStringCmdCfg[iLineCfg]), SIZEOF(arStringCmdCfg[iLineCfg]) ,	ADR(strTemp));
					IL_CONCAT(ADR(asStringCmdCfg[iLineCfg]), ADR(sTemp2), ADR(asStringCmdCfg[iLineCfg]), SIZEOF(asStringCmdCfg[iLineCfg]));
					sTemp2 :=  ', DeactModule = ';
					//strConcat(ADR	(arStringCmdCfg[iLineCfg]), SIZEOF(arStringCmdCfg[iLineCfg]) ,	ADR(strTemp));
					IL_CONCAT(ADR(asStringCmdCfg[iLineCfg]), ADR(sTemp2), ADR(asStringCmdCfg[iLineCfg]), SIZEOF(asStringCmdCfg[iLineCfg]));
					FOR j := 1 TO iMAX_MODULE_ON_SERCOS_IO DO
						IF NOT refastSercosIOCmdConfig[i].astIOModule[j].bActive AND refastSercosIOCmdConfig[i].astIOModule[j].bConfigured  THEN
							IF bWriteThisLine THEN
								sTemp2 :=  ', ';
								//strConcat(ADR	(arStringCmdCfg[iLineCfg]), SIZEOF(arStringCmdCfg[iLineCfg]) ,	ADR(strTemp));
								IL_CONCAT(ADR(asStringCmdCfg[iLineCfg]), ADR(sTemp2), ADR(asStringCmdCfg[iLineCfg]), SIZEOF(asStringCmdCfg[iLineCfg]));
							END_IF	
							sTemp2 := INT_TO_STRING (j);
							//strConcat(ADR	(arStringCmdCfg[iLineCfg]), SIZEOF(arStringCmdCfg[iLineCfg]) ,	ADR(strTemp));
							IL_CONCAT(ADR(asStringCmdCfg[iLineCfg]), ADR(sTemp2), ADR(asStringCmdCfg[iLineCfg]), SIZEOF(asStringCmdCfg[iLineCfg]));
							
							bWriteThisLine := TRUE;
						END_IF
					END_FOR
				
					
					IF NOT bWriteThisLine THEN
						sTemp2 := 	asStringCmdCfg[iLineCfg];
						asStringCmdCfg[iLineCfg] := '; ';
						//strConcat(ADR (arStringCmdCfg[iLineCfg]), SIZEOF(arStringCmdCfg[iLineCfg]) ,ADR(strTemp));
						IL_CONCAT(ADR(asStringCmdCfg[iLineCfg]), ADR(sTemp2), ADR(asStringCmdCfg[iLineCfg]), SIZEOF(asStringCmdCfg[iLineCfg]));
					END_IF
					
					IF NOT (asStringCmdCfg[iLineCfg]= asStringActCfg[iLineCfg]) THEN
						OUT_bReboot := TRUE;
					END_IF
					iLineCfg := iLineCfg +1; 	// next line
						
				ELSE
					// deactivate complete sercos slave			
					asStringCmdCfg[iLineCfg] := '';
								
					sTemp2 := 'SlaveDeactAddr = ';
					//strConcat(ADR	(arStringCmdCfg[iLineCfg]), SIZEOF(arStringCmdCfg[iLineCfg]) ,	ADR(strTemp));
					IL_CONCAT(ADR(asStringCmdCfg[iLineCfg]), ADR(sTemp2), ADR(asStringCmdCfg[iLineCfg]), SIZEOF(asStringCmdCfg[iLineCfg]));
					sTemp2 := INT_TO_STRING (refastSercosIOCmdConfig[i].iSercosAddress);
					//strConcat(ADR	(arStringCmdCfg[iLineCfg]), SIZEOF(arStringCmdCfg[iLineCfg]) ,	ADR(strTemp));
					IL_CONCAT(ADR(asStringCmdCfg[iLineCfg]), ADR(sTemp2), ADR(asStringCmdCfg[iLineCfg]), SIZEOF(asStringCmdCfg[iLineCfg]));
	
					IF NOT (asStringCmdCfg[iLineCfg]= asStringActCfg[iLineCfg]) THEN
						OUT_bReboot := TRUE;
					END_IF
				
					iLineCfg := iLineCfg +1; 	// next line
				END_IF
			ELSIF refastSercosIOCmdConfig[i].iSercosAddress = 0 THEN
				// End LOOP
	 			i := iMAX_SERCOS_IO + 1;
			END_IF	
		END_FOR
		
		asStringCmdCfg[iLineCfg] := ';-----------------------------------------';
		iLineCfg := iLineCfg +1;	 	// next line

		asStringCmdCfg[iLineCfg] := '';	
		iLineCfg := iLineCfg +1;	 	// next line
		
		iEOF := iLineCfg -1 ;			//End Of File
		
		IF IN_bWriteSercosIOAddress THEN 
			iState 		:= 290;
		ELSE
			iState 		:= 299;
		END_IF
			

(* ################################################################################ *)	
	// Check all I/Os which are found in C-0-0510 (only address of SIII Buscoupler)
(* ################################################################################ *)			
	290: 			
		j := 1;
		FOR i := 1 TO iMAX_SERCOS_IO DO
			refastSercosIOConfigError[i].bError := FALSE;
			refastSercosIOConfigError[i].iSercosAddress := 0;
			refastSercosIOConfigError[i].sErrorMessage := '';
			IF refastSercosIOCmdConfig[i].bActive THEN
				IF NOT (apiPointerToC510[j] = 0) THEN
					apiPointerToC510[j]^ := refastSercosIOCmdConfig[i].iSercosAddress;
					j := j+1;
				ELSE 
					refastSercosIOConfigError[i].bError := TRUE;
					refastSercosIOConfigError[i].iSercosAddress := refastSercosIOCmdConfig[i].iSercosAddress;;
				
					sTemp2 :='';
					refastSercosIOConfigError[i].sErrorMessage := 'IO ';
					sTemp2 := refastSercosIOCmdConfig[i].sName;
					//strConcat(ADR	(SercosIOConfigError[i].ErrorMessage), (SIZEOF(SercosIOConfigError[i].ErrorMessage)) ,	ADR(strTemp));
					IL_CONCAT(ADR(refastSercosIOConfigError[i].sErrorMessage), ADR(sTemp2), ADR(refastSercosIOConfigError[i].sErrorMessage), SIZEOF(refastSercosIOConfigError[i].sErrorMessage));
					sTemp2 := ' with sercos address ';
					//strConcat(ADR	(SercosIOConfigError[i].ErrorMessage), (SIZEOF(SercosIOConfigError[i].ErrorMessage)) ,	ADR(strTemp));
					IL_CONCAT(ADR(refastSercosIOConfigError[i].sErrorMessage), ADR(sTemp2), ADR(refastSercosIOConfigError[i].sErrorMessage), SIZEOF(refastSercosIOConfigError[i].sErrorMessage));
					sTemp2 := INT_TO_STRING(refastSercosIOConfigError[i].iSercosAddress);
					//strConcat(ADR	(SercosIOConfigError[i].ErrorMessage), (SIZEOF(SercosIOConfigError[i].ErrorMessage)) ,	ADR(strTemp));
					IL_CONCAT(ADR(refastSercosIOConfigError[i].sErrorMessage), ADR(sTemp2), ADR(refastSercosIOConfigError[i].sErrorMessage), SIZEOF(refastSercosIOConfigError[i].sErrorMessage));
					sTemp2 := ' not found on bus';				
					IL_CONCAT(ADR(refastSercosIOConfigError[i].sErrorMessage), ADR(sTemp2), ADR(refastSercosIOConfigError[i].sErrorMessage), SIZEOF(refastSercosIOConfigError[i].sErrorMessage));
					bErrorTemp := TRUE;
					
					IF sDiagMessageInt = '' THEN
						sDiagMessageInt := refastSercosIOConfigError[i].sErrorMessage;
					END_IF			
					
				END_IF
			END_IF
		END_FOR
		
		IF bErrorTemp THEN  
			OUT_ErrorID := 	RESOURCE_ERROR;
			OUT_ErrorIdent.Table :=	USER1_TABLE;       
			OUT_ErrorIdent.Additional1 := 16#F0003;
			OUT_ErrorIdent.Additional2 := 16#F0000;
			
			iState 		:= 998;
		ELSE
			iState 		:= 295;
		END_IF	
		
(* ################################################################################ *)	
	// Write C-0-0510 (only address of SIII Buscoupler)
(* ################################################################################ *)					
	295:	
		fbWriteListParameter(
			Execute			:= TRUE, 
			ParameterNumber	:= GVL_C_Param_ID.FP_C_0_0510, 
			NoOfBytes		:= uiLengthArC510, 
			ValueAdr		:= ADR(aiC510), 
			Axis			:= NoAxis );
				
		IF fbWriteListParameter.Done THEN
			fbWriteListParameter(Execute	:= FALSE,
								Axis	:= NoAxis);
			iState 	:= 299;
			i		:= 0;
		ELSIF fbWriteListParameter.Error THEN
			OUT_ErrorID 	:= fbWriteListParameter.ErrorID;
			OUT_ErrorIdent 	:= fbWriteListParameter.ErrorIdent;
			fbWriteListParameter(Execute	:= FALSE,
								Axis	:= NoAxis);
			iState 		:= 998;
		END_IF
	
		
(* ################################################################################ *)	
	// End
(* ################################################################################ *)					
	299:
		iState := 300;		

END_CASE
END_METHOD

METHOD M_3ConfigInlineIO : BOOL

CASE iState OF		
					
	300:
		M_DelStructure(ADR(refastInlineIOConfigError), SIZEOF(refastInlineIOConfigError));
		IF IN_bCheckInlineIOConfig THEN
			iState := 310;
		ELSIF IN_bConfigInlineIO THEN
			iState := 350;
		ELSE
			iState := 399;
		END_IF

(* ################################################################################ *)	
	// Check if Configuration is OK
(* ################################################################################ *)			
	310:
		k:= 1;
		FOR i := 1 TO iMAX_INLINE_IO DO
			IF refastInlineIOActConfig[i].bAvailable THEN	
				refastInlineIOConfigError[i].bIOFoundAndNotConfigured := TRUE;
				refastInlineIOConfigError[i].sName := '';
	
				FOR j := k TO iMAX_INLINE_IO DO
					IF refastInlineIOActConfig[i].bAvailable AND refastInlineIOCmdConfig[j].bActive AND refastInlineIOCmdConfig[j].bConfigured THEN 
						// Wrong IO Type
						IF NOT (refastInlineIOActConfig[i].eIOType = refastInlineIOCmdConfig[j].eIOType) THEN
							refastInlineIOConfigError[i].bWrongIOType := TRUE;
							refastInlineIOConfigError[i].sName := refastInlineIOCmdConfig[j].sName;
						END_IF
						k := j+1;									// save index 
						refastInlineIOConfigError[i].bIOFoundAndNotConfigured := FALSE;
						j := iMAX_SERCOS_IO +1; 		// End LOOP
					END_IF	
				END_FOR
			ELSE	
				i := 	iMAX_SERCOS_IO +1;  // End LOOP
			END_IF	
		END_FOR

	// Are there still some IO configured which where not found on the Inline Bus?
		IF k <= iMAX_INLINE_IO THEN
			FOR j := k TO iMAX_INLINE_IO DO
				IF refastInlineIOCmdConfig[j].bActive THEN
 					refastInlineIOConfigError[j].bIOConfiguredAndNotFound := TRUE;
					refastInlineIOConfigError[j].sName := refastInlineIOCmdConfig[j].sName;
				END_IF
			END_FOR
		END_IF	
	
		iState := 320;
		
(* ################################################################################ *)	
	// generate Error if necessary 
(* ################################################################################ *)	
	320:
		FOR i := 1 TO iMAX_INLINE_IO DO
			IF refastInlineIOConfigError[i].bWrongIOType	
				OR refastInlineIOConfigError[i].bIOFoundAndNotConfigured 
				OR refastInlineIOConfigError[i].bIOConfiguredAndNotFound THEN
					refastInlineIOConfigError[i].bError := TRUE;
									
					bErrorTemp := TRUE;
									
					// Create Error Message
					refastInlineIOConfigError[i].sErrorMessage := 'Inline IO ';
					sTemp2 := refastInlineIOConfigError[i].sName ;
					//strConcat(ADR	(InlineIOConfigError[i].ErrorMessage), SIZEOF(SercosIOConfigError[i].ErrorMessage) ,	ADR(strTemp));
					IL_CONCAT(ADR(refastInlineIOConfigError[i].sErrorMessage), ADR(sTemp2), ADR(refastInlineIOConfigError[i].sErrorMessage), SIZEOF(refastSercosIOConfigError[i].sErrorMessage));
					sTemp2 :=  ' Slot '; ;
					//strConcat(ADR	(InlineIOConfigError[i].ErrorMessage), SIZEOF(InlineIOConfigError[i].ErrorMessage) ,	ADR(strTemp));
					IL_CONCAT(ADR(refastInlineIOConfigError[i].sErrorMessage), ADR(sTemp2), ADR(refastInlineIOConfigError[i].sErrorMessage), SIZEOF(refastSercosIOConfigError[i].sErrorMessage));
					sTemp2 := INT_TO_STRING(i);
					//strConcat(ADR	(InlineIOConfigError[i].ErrorMessage), SIZEOF(InlineIOConfigError[i].ErrorMessage) ,	ADR(strTemp));
					IL_CONCAT(ADR(refastInlineIOConfigError[i].sErrorMessage), ADR(sTemp2), ADR(refastInlineIOConfigError[i].sErrorMessage), SIZEOF(refastSercosIOConfigError[i].sErrorMessage));
					sTemp2 := ' shows error: ';
					//strConcat(ADR	(InlineIOConfigError[i].ErrorMessage), SIZEOF(InlineIOConfigError[i].ErrorMessage) ,	ADR(strTemp));
					IL_CONCAT(ADR(refastInlineIOConfigError[i].sErrorMessage), ADR(sTemp2), ADR(refastInlineIOConfigError[i].sErrorMessage), SIZEOF(refastSercosIOConfigError[i].sErrorMessage));
					sTemp2 :='';
					IF refastInlineIOConfigError[i].bWrongIOType	THEN
						sTemp2 :='wrong IO Type';
						//strConcat(ADR	(InlineIOConfigError[i].ErrorMessage), SIZEOF(InlineIOConfigError[i].ErrorMessage) ,	ADR(strTemp));
						IL_CONCAT(ADR(refastInlineIOConfigError[i].sErrorMessage), ADR(sTemp2), ADR(refastInlineIOConfigError[i].sErrorMessage), SIZEOF(refastSercosIOConfigError[i].sErrorMessage));
						sTemp2 :=', ';
					END_IF
					
					IF refastInlineIOConfigError[i].bIOConfiguredAndNotFound	THEN
						//strConcat(ADR	(InlineIOConfigError[i].ErrorMessage), SIZEOF(InlineIOConfigError[i].ErrorMessage) ,	ADR(strTemp));
						IL_CONCAT(ADR(refastInlineIOConfigError[i].sErrorMessage), ADR(sTemp2), ADR(refastInlineIOConfigError[i].sErrorMessage), SIZEOF(refastSercosIOConfigError[i].sErrorMessage));
						sTemp2 :='configured but not found';
						//strConcat(ADR	(InlineIOConfigError[i].ErrorMessage), SIZEOF(InlineIOConfigError[i].ErrorMessage) ,	ADR(strTemp));
						IL_CONCAT(ADR(refastInlineIOConfigError[i].sErrorMessage), ADR(sTemp2), ADR(refastInlineIOConfigError[i].sErrorMessage), SIZEOF(refastSercosIOConfigError[i].sErrorMessage));
						sTemp2 :=', ';
					END_IF
					
					IF refastInlineIOConfigError[i].bIOFoundAndNotConfigured	THEN
						//strConcat(ADR	(InlineIOConfigError[i].ErrorMessage), SIZEOF(InlineIOConfigError[i].ErrorMessage) ,	ADR(strTemp));
						IL_CONCAT(ADR(refastInlineIOConfigError[i].sErrorMessage), ADR(sTemp2), ADR(refastInlineIOConfigError[i].sErrorMessage), SIZEOF(refastSercosIOConfigError[i].sErrorMessage));
						sTemp2 :='found but not configured in DeviceCmdConfig';
						//strConcat(ADR	(InlineIOConfigError[i].ErrorMessage), SIZEOF(InlineIOConfigError[i].ErrorMessage) ,	ADR(strTemp));
						IL_CONCAT(ADR(refastInlineIOConfigError[i].sErrorMessage), ADR(sTemp2), ADR(refastInlineIOConfigError[i].sErrorMessage), SIZEOF(refastSercosIOConfigError[i].sErrorMessage));
						sTemp2 :=', ';
					END_IF	
					
					ML_SetDiagEntry(
						Severity:= enSeverity, 
						Class:= enClass, 
						Facility:= E_LOG_FACILITY.USER, 
						Code:= wDIAG_CODE, 
						Text:= ADR(refastInlineIOConfigError[i].sErrorMessage));
					
					IF sDiagMessageInt = '' THEN
						sDiagMessageInt := refastInlineIOConfigError[i].sErrorMessage;
					END_IF			
						
			END_IF
		END_FOR
			
		IF bErrorTemp THEN  
			OUT_ErrorID := 	RESOURCE_ERROR;
			OUT_ErrorIdent.Table :=	USER1_TABLE;       
			OUT_ErrorIdent.Additional1 := 16#F0005;
			OUT_ErrorIdent.Additional2 := 16#F0000;

			iState 		:= 998;
		ELSIF IN_bConfigInlineIO THEN
			iState 		:= 350;
		ELSE	
			iState 		:= 399;
		END_IF		
	
			
(* ################################################################################ *)	
	// create String for UserDefs.cfg
(* ################################################################################ *)				
	350:
		(* Example:
	;---------- Master.0 ----------
	[InlineIO.Master.0]
	ModuleDeactPosi = 3
	ModuleDeactPosi = 7
	ModuleDeactPosi = 15
	ModuleDeactPosi = 16
	;------------------------------

		*)

		//	Header
		asStringCmdCfg[iLineCfg] := ';--------------- Inline IO --------------- ';
		iLineCfg := iLineCfg + 1;	 	// next line
		asStringCmdCfg[iLineCfg] := '[InlineIO.Master.0]'	;
		iLineCfg := iLineCfg +1;	 	// next line
		
		FOR i := 1 TO iMAX_INLINE_IO DO
			IF refastInlineIOCmdConfig[i].bConfigured THEN 
				IF refastInlineIOCmdConfig[i].bActive THEN
					asStringCmdCfg[iLineCfg] := '; ';
				ELSE			
					asStringCmdCfg[iLineCfg] := '';
				END_IF	
				
				sTemp2 := 'ModuleDeactPosi = ';
				//strConcat(ADR	(arStringCmdCfg[iLineCfg]), SIZEOF(arStringCmdCfg[iLineCfg]) ,	ADR(strTemp));
				IL_CONCAT(ADR	(asStringCmdCfg[iLineCfg]), ADR(sTemp2), ADR	(asStringCmdCfg[iLineCfg]), SIZEOF(asStringCmdCfg[iLineCfg]));
				sTemp2 := INT_TO_STRING (i);
				//strConcat(ADR	(arStringCmdCfg[iLineCfg]), SIZEOF(arStringCmdCfg[iLineCfg]) ,	ADR(strTemp));
				IL_CONCAT(ADR	(asStringCmdCfg[iLineCfg]), ADR(sTemp2), ADR	(asStringCmdCfg[iLineCfg]), SIZEOF(asStringCmdCfg[iLineCfg]));
				
				IF NOT (asStringCmdCfg[iLineCfg] = asStringActCfg[iLineCfg]) THEN
					OUT_bReboot := TRUE;
				END_IF
			
				iLineCfg := iLineCfg +1; 	// next line
				
			ELSIF NOT refastInlineIOCmdConfig[i].bConfigured  THEN
				// End LOOP
	 			i := iMAX_INLINE_IO + 1;	
			END_IF	
			
			
		END_FOR
		
		asStringCmdCfg[iLineCfg] := ';-----------------------------------------'	;
		iLineCfg := iLineCfg +1;	 	// next line

		asStringCmdCfg[iLineCfg] := ''	;
		iLineCfg := iLineCfg +1;	 	// next line
		
		iEOF := iLineCfg -1 ;			//End Of File
		iState := 399;
		
(* ################################################################################ *)	
	// End
(* ################################################################################ *)					
	399:
		iState := 400;		

END_CASE
END_METHOD

METHOD M_4ConfigProfibsIO : BOOL


CASE iState OF		
(* ################################################################################ *)	
	// create String for UserDefs.cfg
(* ################################################################################ *)						
	400:
		IF IN_bConfigProfibusIO THEN
			iState := 410;
		ELSE
			iState := 499;
		END_IF

	410:
		(* Example:
		; *****************************
		; Onboard Master
		; *****************************
		
		[ProfibusDP.Master.0]
		SlaveDeactAddr = 5
		SlaveDeactAddr = 8
		SlaveDeactAddr = 25
		
		
		; *******************************
		; Master auf einem Funktionsmodul
		; *******************************
		
		[ProfibusDP.Master.1]
		SlaveDeactAddr = 64
		SlaveDeactAddr = 30
		SlaveDeactAddr = 112
		SlaveDeactAddr = 3
	*)

		//	Header

		asStringCmdCfg[iLineCfg] := ';--------------- PROFINET IO --------------- ';
		iLineCfg := iLineCfg + 1;	 	// next line
		
		FOR j := 1 TO iMAX_PROFIBUS_MASTER DO
//			IF ProfibusIOCmdConfig[j,0].Active THEN			// Master is active
				asStringCmdCfg[iLineCfg] := '[ProfibusDP.Master.';
				sTemp2 := INT_TO_STRING(j-1);
				//strConcat(ADR	(arStringCmdCfg[iLineCfg]), SIZEOF(arStringCmdCfg[iLineCfg]) ,	ADR(strTemp));
				IL_CONCAT(ADR(asStringCmdCfg[iLineCfg]), ADR(sTemp2), ADR(asStringCmdCfg[iLineCfg]), SIZEOF(asStringCmdCfg[iLineCfg]));
				sTemp2 := ']';
				//strConcat(ADR	(arStringCmdCfg[iLineCfg]), SIZEOF(arStringCmdCfg[iLineCfg]) ,	ADR(strTemp));
				IL_CONCAT(ADR(asStringCmdCfg[iLineCfg]), ADR(sTemp2), ADR(asStringCmdCfg[iLineCfg]), SIZEOF(asStringCmdCfg[iLineCfg]));
				
				iLineCfg := iLineCfg +1;	 	// next line
	
				FOR i := 1 TO iMAX_PROFIBUS_SLAVE DO
					IF refastProfibusIOCmdConfig[j,i].iAddress <> 0 THEN 
						IF refastProfibusIOCmdConfig[j,i].bActive THEN
							asStringCmdCfg[iLineCfg] := '; ';
						ELSE			
							asStringCmdCfg[iLineCfg] := '';
						END_IF	
						
						sTemp2 := 'SlaveDeactAddr = ';
						//strConcat(ADR	(arStringCmdCfg[iLineCfg]), SIZEOF(arStringCmdCfg[iLineCfg]) ,	ADR(strTemp));
						IL_CONCAT(ADR(asStringCmdCfg[iLineCfg]), ADR(sTemp2), ADR(asStringCmdCfg[iLineCfg]), SIZEOF(asStringCmdCfg[iLineCfg]));
						sTemp2 := INT_TO_STRING (refastProfibusIOCmdConfig[j,i].iAddress);
						//strConcat(ADR	(arStringCmdCfg[iLineCfg]), SIZEOF(arStringCmdCfg[iLineCfg]) ,	ADR(strTemp));
						IL_CONCAT(ADR(asStringCmdCfg[iLineCfg]), ADR(sTemp2), ADR(asStringCmdCfg[iLineCfg]), SIZEOF(asStringCmdCfg[iLineCfg]));
						
						IF NOT (asStringCmdCfg[iLineCfg]= asStringActCfg[iLineCfg]) THEN
							OUT_bReboot := TRUE;
						END_IF
					
						iLineCfg := iLineCfg +1; 	// next line
					
					ELSIF refastProfibusIOCmdConfig[j,i].iAddress = 0 THEN
						// End LOOP
	 					i := iMAX_PROFIBUS_SLAVE + 1;	
					END_IF	
					
				
				END_FOR
				
				asStringCmdCfg[iLineCfg] := ';-------------------------------------------'	;
				iLineCfg := iLineCfg +1;	 	// next line
		
				asStringCmdCfg[iLineCfg] := ''	;
				iLineCfg := iLineCfg +1;	 	// next line
				
				iEOF := iLineCfg -1 ;			//End Of File
//			END_IF	
		END_FOR	
		iState := 499;
		
(* ################################################################################ *)	
	// End
(* ################################################################################ *)					
	499:
		iState := 500;		

END_CASE
END_METHOD

METHOD M_5ConfigProfinetIO : BOOL
// Tip von Hr. Kohl: Schritt 550 umsetzen wie Schritt 350 und Fehlerhandling anschließend, wenn Schritt 350 tut.
// Gucken in der Hilfe bei Index "UserDefs.cfg, Profinet IO-Devices / Profinet IO-Module deaktivieren"
// Name: iv2-g500ca-g30f
// 


CASE iState OF		
(* ################################################################################ *)	
	// create String for UserDefs.cfg
(* ################################################################################ *)						
	500:
		IF IN_bConfigPNIO THEN
			iState := 510;
		ELSE
			iState := 599;
		END_IF
	

	510:
		(* Example:
        ;**************************************************
		;---------- PROFINET IO ----------
		;**************************************************
		[PROFINETIO.Controller.0]
		
		DeviceDeactName = myDeviceName12
		DeviceName = myDeviceName14, DeactModule=2,3
		*)

		//	Header

		asStringCmdCfg[iLineCfg] := ';--------------- PROFINET IO --------------- ';
		iLineCfg := iLineCfg + 1;	 	// next line
		
		FOR j := 1 TO iMAX_PN_MASTER DO
	
			IF (refastPNIOCmdConfig[j,1].sPNDeviceName <> '') THEN			// at least one device is configured
				asStringCmdCfg[iLineCfg] := '[PROFINETIO.Controller.';
				sTemp2 := INT_TO_STRING(j-1);
				//strConcat(ADR	(arStringCmdCfg[iLineCfg]), SIZEOF(arStringCmdCfg[iLineCfg]) ,	ADR(strTemp));
				IL_CONCAT(ADR(asStringCmdCfg[iLineCfg]), ADR(sTemp2), ADR(asStringCmdCfg[iLineCfg]), SIZEOF(asStringCmdCfg[iLineCfg]));
				sTemp2 := ']';
				//strConcat(ADR	(arStringCmdCfg[iLineCfg]), SIZEOF(arStringCmdCfg[iLineCfg]) ,	ADR(strTemp));
				IL_CONCAT(ADR(asStringCmdCfg[iLineCfg]), ADR(sTemp2), ADR(asStringCmdCfg[iLineCfg]), SIZEOF(asStringCmdCfg[iLineCfg]));
				
				iLineCfg := iLineCfg +1;	 	// next line
		
				FOR i := 1 TO iMAX_PN_SLAVE DO
					IF refastPNIOCmdConfig[j,i].sPNDeviceName <> '' THEN 
						IF refastPNIOCmdConfig[j,i].bActive THEN
							// deactivate only modules
							//arStringCmdCfg[iLineCfg] := '; ';
							
							asStringCmdCfg[iLineCfg] := '';
							bWriteThisLine := FALSE;
							sTemp2 := 'DeviceName = ';
							//strConcat(ADR	(arStringCmdCfg[iLineCfg]), SIZEOF(arStringCmdCfg[iLineCfg]) ,	ADR(strTemp));
							IL_CONCAT(ADR(asStringCmdCfg[iLineCfg]), ADR(sTemp2), ADR(asStringCmdCfg[iLineCfg]), SIZEOF(asStringCmdCfg[iLineCfg]));
							sTemp2 := (refastPNIOCmdConfig[j,i].sPNDeviceName);
							//strConcat(ADR	(arStringCmdCfg[iLineCfg]), SIZEOF(arStringCmdCfg[iLineCfg]) ,	ADR(strTemp));
							IL_CONCAT(ADR(asStringCmdCfg[iLineCfg]), ADR(sTemp2), ADR(asStringCmdCfg[iLineCfg]), SIZEOF(asStringCmdCfg[iLineCfg]));
							sTemp2 :=  ', DeactModule = ';
							//strConcat(ADR	(arStringCmdCfg[iLineCfg]), SIZEOF(arStringCmdCfg[iLineCfg]) ,	ADR(strTemp));
							IL_CONCAT(ADR(asStringCmdCfg[iLineCfg]), ADR(sTemp2), ADR(asStringCmdCfg[iLineCfg]), SIZEOF(asStringCmdCfg[iLineCfg]));
							FOR k := 1 TO iMAX_MODULE_ON_PN_IO DO
								IF NOT refastPNIOCmdConfig[j,i].astIOModule[k].bActive AND refastPNIOCmdConfig[j,i].astIOModule[k].bConfigured  THEN
									IF bWriteThisLine THEN
										sTemp2 :=  ', ';
										//strConcat(ADR	(arStringCmdCfg[iLineCfg]), SIZEOF(arStringCmdCfg[iLineCfg]) ,	ADR(strTemp));
										IL_CONCAT(ADR(asStringCmdCfg[iLineCfg]), ADR(sTemp2), ADR(asStringCmdCfg[iLineCfg]), SIZEOF(asStringCmdCfg[iLineCfg]));
									END_IF	
									sTemp2 := INT_TO_STRING (k);
									//strConcat(ADR	(arStringCmdCfg[iLineCfg]), SIZEOF(arStringCmdCfg[iLineCfg]) ,	ADR(strTemp));
									IL_CONCAT(ADR(asStringCmdCfg[iLineCfg]), ADR(sTemp2), ADR(asStringCmdCfg[iLineCfg]), SIZEOF(asStringCmdCfg[iLineCfg]));
									
									bWriteThisLine := TRUE;
								END_IF
							END_FOR
						
							
							IF NOT bWriteThisLine THEN
								sTemp2 := 	asStringCmdCfg[iLineCfg];
								asStringCmdCfg[iLineCfg] := '; ';
								//strConcat(ADR (arStringCmdCfg[iLineCfg]), SIZEOF(arStringCmdCfg[iLineCfg]) ,ADR(strTemp));
								IL_CONCAT(ADR(asStringCmdCfg[iLineCfg]), ADR(sTemp2), ADR(asStringCmdCfg[iLineCfg]), SIZEOF(asStringCmdCfg[iLineCfg]));
							END_IF
							
							IF NOT (asStringCmdCfg[iLineCfg]= asStringActCfg[iLineCfg]) THEN
								OUT_bReboot := TRUE;
							END_IF
							iLineCfg := iLineCfg +1; 	// next line
								
						ELSE			
							asStringCmdCfg[iLineCfg] := '';
							sTemp2 := 'DeviceDeactName = ';
							//strConcat(ADR	(arStringCmdCfg[iLineCfg]), SIZEOF(arStringCmdCfg[iLineCfg]) ,	ADR(strTemp));
							IL_CONCAT(ADR(asStringCmdCfg[iLineCfg]), ADR(sTemp2), ADR(asStringCmdCfg[iLineCfg]), SIZEOF(asStringCmdCfg[iLineCfg]));
							sTemp2 := (refastPNIOCmdConfig[j,i].sPNDeviceName);
							//strConcat(ADR	(arStringCmdCfg[iLineCfg]), SIZEOF(arStringCmdCfg[iLineCfg]) ,	ADR(strTemp));
							IL_CONCAT(ADR(asStringCmdCfg[iLineCfg]), ADR(sTemp2), ADR(asStringCmdCfg[iLineCfg]), SIZEOF(asStringCmdCfg[iLineCfg]));
							
							IF NOT (asStringCmdCfg[iLineCfg]= asStringActCfg[iLineCfg]) THEN
								OUT_bReboot := TRUE;
							END_IF
						
							iLineCfg := iLineCfg +1; 	// next line
						END_IF	
					ELSIF refastPNIOCmdConfig[j,i].sPNDeviceName = '' THEN
						// End LOOP
						i := iMAX_PN_SLAVE + 1;	
					END_IF	
					
				END_FOR
				
				asStringCmdCfg[iLineCfg] := ';-------------------------------------------'	;
				iLineCfg := iLineCfg +1;	 	// next line
		
				asStringCmdCfg[iLineCfg] := ''	;
				iLineCfg := iLineCfg +1;	 	// next line
				
				iEOF := iLineCfg -1 ;			//End Of File
			END_IF	
		END_FOR	
		iState := 599;
	
(* ################################################################################ *)	
	// End
(* ################################################################################ *)					
	599:
		iState := 800;		

END_CASE
END_METHOD

METHOD M_8WriteConfig : BOOL


CASE iState OF
(* ################################################################################ *)	
	// Open File UserDefs.cfg
(* ################################################################################ *)	
	800: // DevicePlcAdd.new neu anlegen und zum schreiben öffnen
		hCfg := SysFileStreamFOpenV3(sFileAndPathInt, 'w');
		iState :=810;

(* ################################################################################ *)	
	// Write into File 
(* ################################################################################ *)		
	810:
		FOR i := 1 TO iEOF DO
			diResult := FUN_WriteLnString(hCfg, asStringCmdCfg[i]);	// M_WriteLnString(hCfg, asStringCmdCfg[i]);  	
		END_FOR
		iState :=820;

(* ################################################################################ *)	
	// Close File UserDefs.cfg
(* ################################################################################ *)	
	820:
		SysFileStreamFClose(hCfg);
		iState :=899;
	
(* ################################################################################ *)	
	// End
(* ################################################################################ *)
	899: 
		iState := 900;

END_CASE
END_METHOD

METHOD M_9ErrorDone : BOOL
CASE iState OF
	
(* ################################################################################ *)	
	// Reboot necessary?
(* ################################################################################ *)			
	900:
		IF OUT_bReboot AND IN_bRebootAuto THEN
			IMCCtrl.Admin._OpMode := IMC_MODE_CTRL_P0;
			IF IMCSTatus.Admin.ModeStatus_P0 AND NOT IMCSTatus.Admin.PhaseSwitchActive THEN
				fbCommand(	Execute			:= TRUE, 
					ParameterNumber	:= GVL_C_Param_ID.FP_C_0_1021, 
					Axis			:= NoAxis);
			END_IF
			MB_IMCInterface();
		ELSE
			iState := 910;		
		END_IF
		
(* ################################################################################ *)	
	//Refresh FP_C_0_0479
(* ################################################################################ *)			
	910:
		fbCommand(	Execute			:= TRUE, 
					ParameterNumber	:= GVL_C_Param_ID.FP_C_0_1009, 
					Axis			:= NoAxis);
		
		IF fbCommand.Done THEN
			fbCommand(	Execute	:= FALSE,
						Axis	:= NoAxis);
			iState	:= 990;
		ELSIF fbCommand.Error THEN
			OUT_ErrorID		:= fbCommand.ErrorID;
			OUT_ErrorIdent	:= fbCommand.ErrorIdent;
			fbCommand(	Execute:= FALSE,
						Axis:= NoAxis);
			iState 		:= 998;
		END_IF	
		
(* ################################################################################ *)	
	// Change sercos reaction back to desired value
(* ################################################################################ *)	
//920:
//	IF UpdateFirmware THEN
//		IF (NOT SercosErrorReaction.F2_Error AND NOT SercosErrorReaction.F5_Error AND NOT SercosErrorReaction.F8_Error)
//			OR SercosErrorReaction.F8_Error THEN
//			dwC506.0 := FALSE;		
//			dwC506.1 := FALSE;
//		ELSIF SercosErrorReaction.F5_Error THEN
//			dwC506.0 := TRUE;
//			dwC506.1 := FALSE;
//		ELSIF SercosErrorReaction.F2_Error THEN  
//			dwC506.0 := FALSE;
//			dwC506.1 := TRUE;	
//		END_IF
//		
//		dwC506.7 := SercosErrorReaction.NoRedundancyWarning;
//		dwC506.8 := SercosErrorReaction.AutoRingRecovery; 
//		
//		fbWriteC506(
//			Execute:=TRUE , 
//			Done=> , 
//			Active=> , 
//			Error=> , 
//			ErrorID=> , 
//			ErrorIdent=> , 
//			ParameterNumber:= FP_C_0_0506, 
//			Value:= 	dwC506, 
//			Axis:= 	NoAxis);
//	END_IF
//	IF fbWriteC506.Done OR NOT UpdateFirmware THEN
//		fbWriteC506(Execute:=FALSE, 
//				Axis:= 	NoAxis);	
//		iState 	:= 990;		
//	ELSIF fbWriteC506.Error THEN
//		ErrorID 	:= fbWriteC506.ErrorID;
//		ErrorIdent 	:= fbWriteC506.ErrorIdent;
//		fbWriteC506(Execute:=FALSE, 
//					Axis:= 	NoAxis);	
//		iState 		:= 998;
//	END_IF		
			
(* ################################################################################ *)	
	// Done
(* ################################################################################ *)	
	990: 			
		OUT_bDone := TRUE;
		OUT_bError := FALSE;
		OUT_bActive := FALSE;
		bErrorTemp := FALSE;
		OUT_sDiagMessage := '';
		
		IF NOT IN_bExecute THEN
			iState := 0;
		END_IF

(* ################################################################################ *)	
	// Change sercos reaction back to desired value
(* ################################################################################ *)	
998:
	iState 	:= 999;		

//	IF UpdateFirmware THEN
//		IF (NOT SercosErrorReaction.F2_Error AND NOT SercosErrorReaction.F5_Error AND NOT SercosErrorReaction.F8_Error)
//			OR SercosErrorReaction.F8_Error THEN
//			dwC506.0 := FALSE;		
//			dwC506.1 := FALSE;
//		ELSIF SercosErrorReaction.F5_Error THEN
//			dwC506.0 := TRUE;
//			dwC506.1 := FALSE;
//		ELSIF SercosErrorReaction.F2_Error THEN  
//			dwC506.0 := FALSE;
//			dwC506.1 := TRUE;	
//		END_IF
//		
//		dwC506.7 := SercosErrorReaction.NoRedundancyWarning;
//		dwC506.8 := SercosErrorReaction.AutoRingRecovery; 
//	
//		fbWriteC506(
//			Execute:=TRUE , 
//			Done=> , 
//			Active=> , 
//			Error=> , 
//			ErrorID=> , 
//			ErrorIdent=> , 
//			ParameterNumber:= FP_C_0_0506, 
//			Value:= 	dwC506, 
//			Axis:= 	NoAxis);
//	END_IF
//	
//	IF fbWriteC506.Done OR fbWriteC506.Error
//	OR NOT UpdateFirmware THEN
//		fbWriteC506(Execute:=FALSE, 
//				Axis:= 	NoAxis);	
//		iState 	:= 999;		
//	END_IF		
							
		
(* ################################################################################ *)	
	// Error
(* ################################################################################ *)	
	999: 			
		IF sDiagMessageInt = '' THEN
			OUT_sDiagMessage := 'Internal FB Error. Check ErrorID and ErrorIdent'; 	
		ELSIF OUT_bActive THEN		// only first cycle 
			OUT_sDiagMessage := sDiagMessageInt;
		END_IF	
		
		OUT_bDone := FALSE;
		OUT_bError := TRUE;
		bErrorTemp := FALSE;
		OUT_bActive := FALSE;
	
		IF NOT IN_bExecute THEN
			iState := 0;
		END_IF
		
END_CASE
END_METHOD

METHOD PRIVATE M_DelStructure : BOOL
VAR_INPUT
	IN_pbToElement: POINTER TO BYTE;
	IN_uiNoOfByte: UINT;
END_VAR
VAR
	i: INT;
END_VAR

FOR i := 1 TO (UINT_TO_INT (IN_uiNoOfByte)) DO
	IN_pbToElement^:= 0;
	IN_pbToElement := IN_pbToElement +1;
END_FOR
END_METHOD

METHOD M_Execute
(*
IF IN_bExecute AND NOT bExecuteOld THEN
	bExecuteOld := TRUE;
	OUT_bActive := TRUE;
	OUT_bDone := FALSE;
	OUT_bError := FALSE;	
	sDiagMessageInt := '';
	OUT_sDiagMessage :='';
	
	// Referenzen aktualisieren
	refastAxesCmdConfig REF= IN_stDeviceCmdConfig.astAxes;
	refastInlineIOCmdConfig REF= IN_stDeviceCmdConfig.astInlineIO;
	refastSercosIOCmdConfig	REF= IN_stDeviceCmdConfig.astSercosIO;
	refastPNIOCmdConfig REF= IN_stDeviceCmdConfig.astPN_IO;
	
	refastAxesActConfig REF= IN_stDeviceActConfig.astAxes;
//	S20IOActConfig REF= DeviceActConfig.S20_IO;
	refastSercosIOActConfig	REF= IN_stDeviceActConfig.astSercosIO;
//	PNIOActConfig REF= DeviceActConfig.PN_IO;
	
	refastAxesConfigError REF= IN_stDeviceConfigError.astAxes;
	refastSercosIOConfigError REF= IN_stDeviceConfigError.astSercosIO;
//	SercosIOCmdConfigError REF= DeviceConfigError.sercos_IO_CmdConfig;
	refastFoundDrivesError REF=	IN_stDeviceConfigError.astFoundDrives;
	refastInlineIOConfigError REF= IN_stDeviceConfigError.astInlineIO;
	
	iState := 10;
ELSIF NOT IN_bExecute AND (OUT_bDone OR OUT_bError) THEN
	bExecuteOld := FALSE;
	OUT_bReboot := FALSE;
	OUT_bActive := FALSE;
	OUT_bDone := FALSE;
	OUT_bError := FALSE;	
	iState := 0;
END_IF

*)

